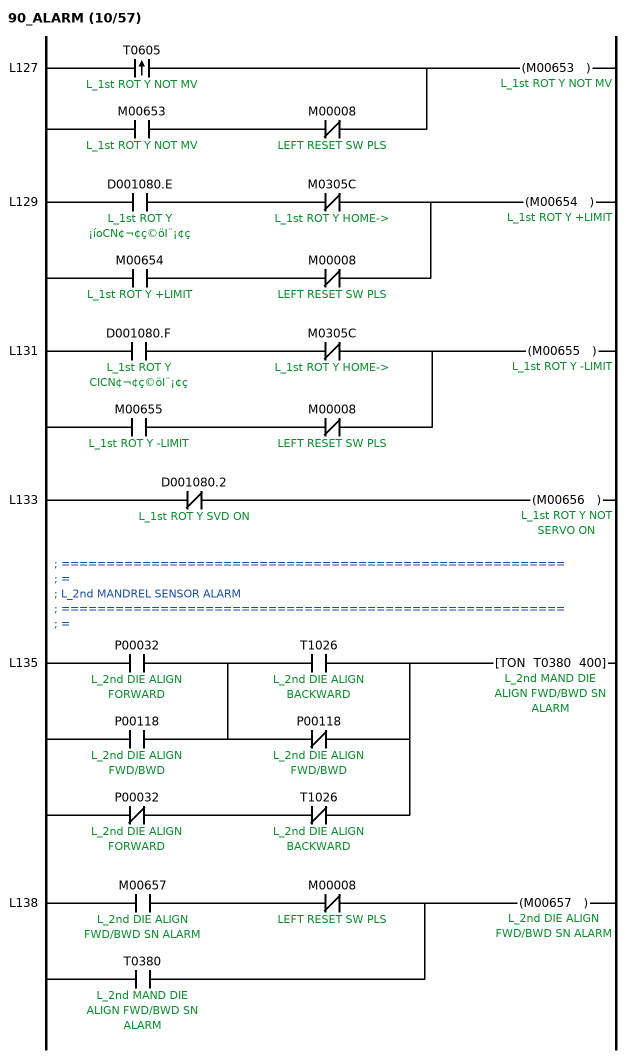
[picture p360: 90_ALARM rungs L127-L138]
; L127
LOADP     T0605	// L_1st ROT Y NOT MV
LOAD      M00653	// L_1st ROT Y NOT MV
AND NOT   M00008	// LEFT RESET SW PLS
OR LOAD
OUT       M00653	// L_1st ROT Y NOT MV
; L129
LOAD      D001080.E	// L_1st ROT Y ¡íoCN¢¬¢ç©öI¨¡¢ç
AND NOT   M0305C	// L_1st ROT Y HOME->
LOAD      M00654	// L_1st ROT Y +LIMIT
AND NOT   M00008	// LEFT RESET SW PLS
OR LOAD
OUT       M00654	// L_1st ROT Y +LIMIT
; L131
LOAD      D001080.F	// L_1st ROT Y CICN¢¬¢ç©öI¨¡¢ç
AND NOT   M0305C	// L_1st ROT Y HOME->
LOAD      M00655	// L_1st ROT Y -LIMIT
AND NOT   M00008	// LEFT RESET SW PLS
OR LOAD
OUT       M00655	// L_1st ROT Y -LIMIT
; L133
LOAD NOT  D001080.2	// L_1st ROT Y SVD ON
OUT       M00656	// L_1st ROT Y NOT SERVO ON
// =========================================================
// 
//        L_2nd MANDREL SENSOR ALARM
// 
// =========================================================
; L135
LOAD      P00032	// L_2nd DIE ALIGN FORWARD
OR        P00118	// L_2nd DIE ALIGN FWD/BWD
LOAD      T1026	// L_2nd DIE ALIGN BACKWARD
OR NOT    P00118	// L_2nd DIE ALIGN FWD/BWD
AND LOAD
LOAD NOT  P00032	// L_2nd DIE ALIGN FORWARD
AND NOT   T1026	// L_2nd DIE ALIGN BACKWARD
OR LOAD
TON       T0380 400	// L_2nd MAND DIE ALIGN FWD/BWD SN ALARM
; L138
LOAD      M00657	// L_2nd DIE ALIGN FWD/BWD SN ALARM
AND NOT   M00008	// LEFT RESET SW PLS
OR        T0380	// L_2nd MAND DIE ALIGN FWD/BWD SN ALARM
OUT       M00657	// L_2nd DIE ALIGN FWD/BWD SN ALARM

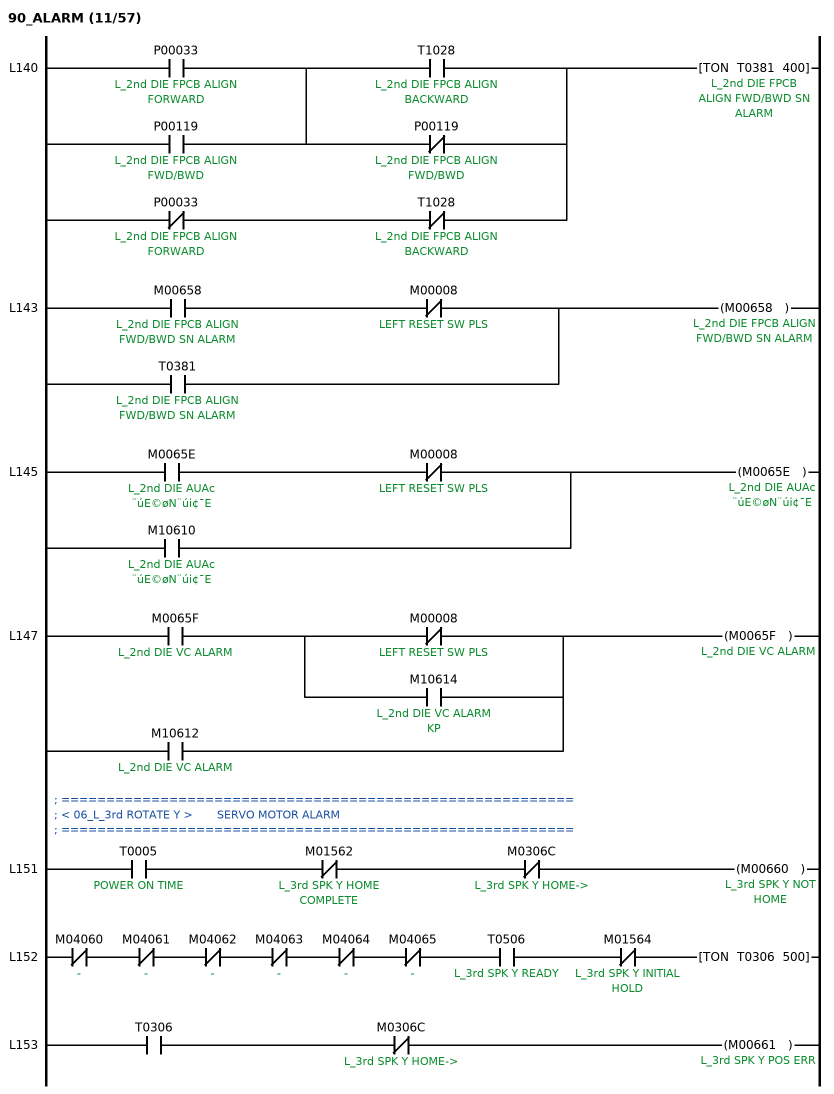
; L140
LOAD      P00033	// L_2nd DIE FPCB ALIGN FORWARD
OR        P00119	// L_2nd DIE FPCB ALIGN FWD/BWD
LOAD      T1028	// L_2nd DIE FPCB ALIGN BACKWARD
OR NOT    P00119	// L_2nd DIE FPCB ALIGN FWD/BWD
AND LOAD
LOAD NOT  P00033	// L_2nd DIE FPCB ALIGN FORWARD
AND NOT   T1028	// L_2nd DIE FPCB ALIGN BACKWARD
OR LOAD
TON       T0381 400	// L_2nd DIE FPCB ALIGN FWD/BWD SN ALARM
; L143
LOAD      M00658	// L_2nd DIE FPCB ALIGN FWD/BWD SN ALARM
AND NOT   M00008	// LEFT RESET SW PLS
OR        T0381	// L_2nd DIE FPCB ALIGN FWD/BWD SN ALARM
OUT       M00658	// L_2nd DIE FPCB ALIGN FWD/BWD SN ALARM
; L145
LOAD      M0065E	// L_2nd DIE AUAc ¨úE©øN¨úi¢¯E
AND NOT   M00008	// LEFT RESET SW PLS
OR        M10610	// L_2nd DIE AUAc ¨úE©øN¨úi¢¯E
OUT       M0065E	// L_2nd DIE AUAc ¨úE©øN¨úi¢¯E
; L147
LOAD      M0065F	// L_2nd DIE VC ALARM
LOAD NOT  M00008	// LEFT RESET SW PLS
OR        M10614	// L_2nd DIE VC ALARM KP
AND LOAD
OR        M10612	// L_2nd DIE VC ALARM
OUT       M0065F	// L_2nd DIE VC ALARM
// =========================================================
// 
//        < 06_L_3rd ROTATE Y >       SERVO MOTOR ALARM
// 
// =========================================================
; L151
LOAD      T0005	// POWER ON TIME
AND NOT   M01562	// L_3rd SPK Y HOME COMPLETE
AND NOT   M0306C	// L_3rd SPK Y HOME->
OUT       M00660	// L_3rd SPK Y NOT HOME
; L152
LOAD NOT  M04060	// -
AND NOT   M04061	// -
AND NOT   M04062	// -
AND NOT   M04063	// -
AND NOT   M04064	// -
AND NOT   M04065	// -
AND       T0506	// L_3rd SPK Y READY
AND NOT   M01564	// L_3rd SPK Y INITIAL HOLD
TON       T0306 500
; L153
LOAD      T0306
AND NOT   M0306C	// L_3rd SPK Y HOME->
OUT       M00661	// L_3rd SPK Y POS ERR

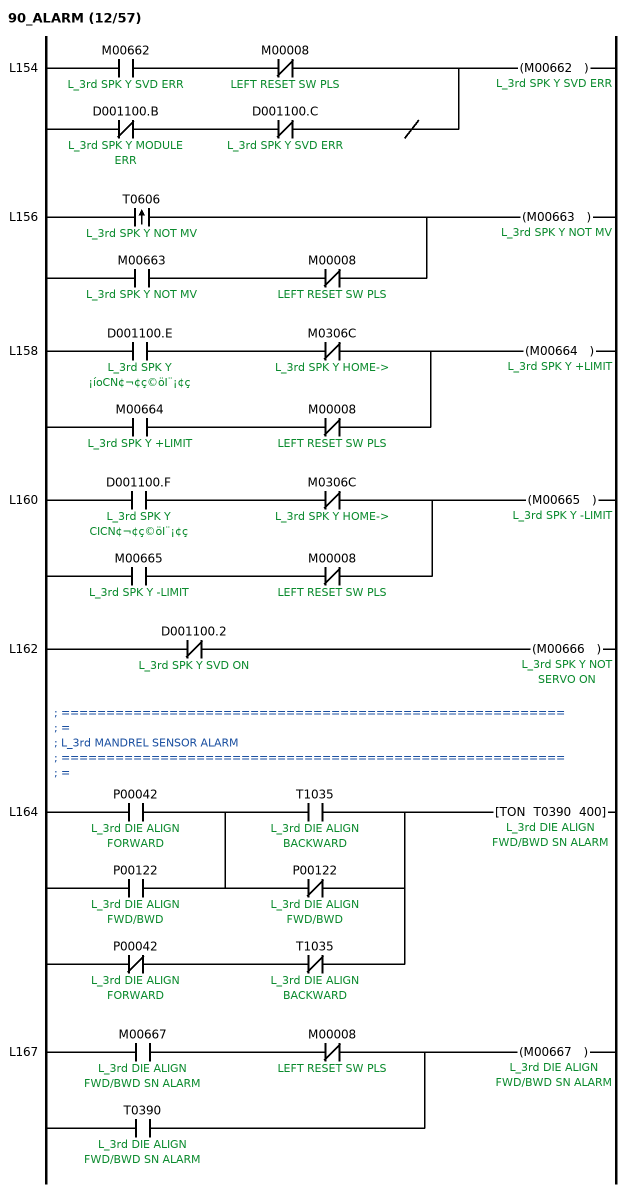
; L154
LOAD      M00662	// L_3rd SPK Y SVD ERR
AND NOT   M00008	// LEFT RESET SW PLS
LOAD NOT  D001100.B	// L_3rd SPK Y MODULE ERR
AND NOT   D001100.C	// L_3rd SPK Y SVD ERR
NOT
OR LOAD
OUT       M00662	// L_3rd SPK Y SVD ERR
; L156
LOADP     T0606	// L_3rd SPK Y NOT MV
LOAD      M00663	// L_3rd SPK Y NOT MV
AND NOT   M00008	// LEFT RESET SW PLS
OR LOAD
OUT       M00663	// L_3rd SPK Y NOT MV
; L158
LOAD      D001100.E	// L_3rd SPK Y ¡íoCN¢¬¢ç©öI¨¡¢ç
AND NOT   M0306C	// L_3rd SPK Y HOME->
LOAD      M00664	// L_3rd SPK Y +LIMIT
AND NOT   M00008	// LEFT RESET SW PLS
OR LOAD
OUT       M00664	// L_3rd SPK Y +LIMIT
; L160
LOAD      D001100.F	// L_3rd SPK Y CICN¢¬¢ç©öI¨¡¢ç
AND NOT   M0306C	// L_3rd SPK Y HOME->
LOAD      M00665	// L_3rd SPK Y -LIMIT
AND NOT   M00008	// LEFT RESET SW PLS
OR LOAD
OUT       M00665	// L_3rd SPK Y -LIMIT
; L162
LOAD NOT  D001100.2	// L_3rd SPK Y SVD ON
OUT       M00666	// L_3rd SPK Y NOT SERVO ON
// =========================================================
// 
//        L_3rd MANDREL SENSOR ALARM
// 
// =========================================================
; L164
LOAD      P00042	// L_3rd DIE ALIGN FORWARD
OR        P00122	// L_3rd DIE ALIGN FWD/BWD
LOAD      T1035	// L_3rd DIE ALIGN BACKWARD
OR NOT    P00122	// L_3rd DIE ALIGN FWD/BWD
AND LOAD
LOAD NOT  P00042	// L_3rd DIE ALIGN FORWARD
AND NOT   T1035	// L_3rd DIE ALIGN BACKWARD
OR LOAD
TON       T0390 400	// L_3rd DIE ALIGN FWD/BWD SN ALARM
; L167
LOAD      M00667	// L_3rd DIE ALIGN FWD/BWD SN ALARM
AND NOT   M00008	// LEFT RESET SW PLS
OR        T0390	// L_3rd DIE ALIGN FWD/BWD SN ALARM
OUT       M00667	// L_3rd DIE ALIGN FWD/BWD SN ALARM

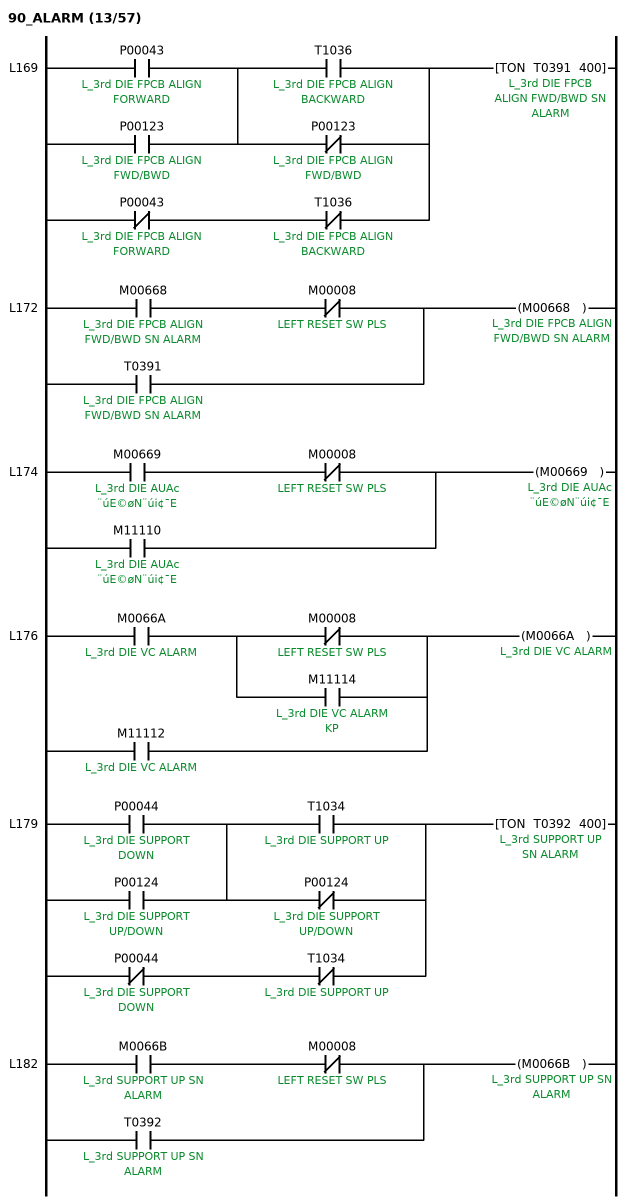
; L169
LOAD      P00043	// L_3rd DIE FPCB ALIGN FORWARD
OR        P00123	// L_3rd DIE FPCB ALIGN FWD/BWD
LOAD      T1036	// L_3rd DIE FPCB ALIGN BACKWARD
OR NOT    P00123	// L_3rd DIE FPCB ALIGN FWD/BWD
AND LOAD
LOAD NOT  P00043	// L_3rd DIE FPCB ALIGN FORWARD
AND NOT   T1036	// L_3rd DIE FPCB ALIGN BACKWARD
OR LOAD
TON       T0391 400	// L_3rd DIE FPCB ALIGN FWD/BWD SN ALARM
; L172
LOAD      M00668	// L_3rd DIE FPCB ALIGN FWD/BWD SN ALARM
AND NOT   M00008	// LEFT RESET SW PLS
OR        T0391	// L_3rd DIE FPCB ALIGN FWD/BWD SN ALARM
OUT       M00668	// L_3rd DIE FPCB ALIGN FWD/BWD SN ALARM
; L174
LOAD      M00669	// L_3rd DIE AUAc ¨úE©øN¨úi¢¯E
AND NOT   M00008	// LEFT RESET SW PLS
OR        M11110	// L_3rd DIE AUAc ¨úE©øN¨úi¢¯E
OUT       M00669	// L_3rd DIE AUAc ¨úE©øN¨úi¢¯E
; L176
LOAD      M0066A	// L_3rd DIE VC ALARM
LOAD NOT  M00008	// LEFT RESET SW PLS
OR        M11114	// L_3rd DIE VC ALARM KP
AND LOAD
OR        M11112	// L_3rd DIE VC ALARM
OUT       M0066A	// L_3rd DIE VC ALARM
; L179
LOAD      P00044	// L_3rd DIE SUPPORT DOWN
OR        P00124	// L_3rd DIE SUPPORT UP/DOWN
LOAD      T1034	// L_3rd DIE SUPPORT UP
OR NOT    P00124	// L_3rd DIE SUPPORT UP/DOWN
AND LOAD
LOAD NOT  P00044	// L_3rd DIE SUPPORT DOWN
AND NOT   T1034	// L_3rd DIE SUPPORT UP
OR LOAD
TON       T0392 400	// L_3rd SUPPORT UP SN ALARM
; L182
LOAD      M0066B	// L_3rd SUPPORT UP SN ALARM
AND NOT   M00008	// LEFT RESET SW PLS
OR        T0392	// L_3rd SUPPORT UP SN ALARM
OUT       M0066B	// L_3rd SUPPORT UP SN ALARM

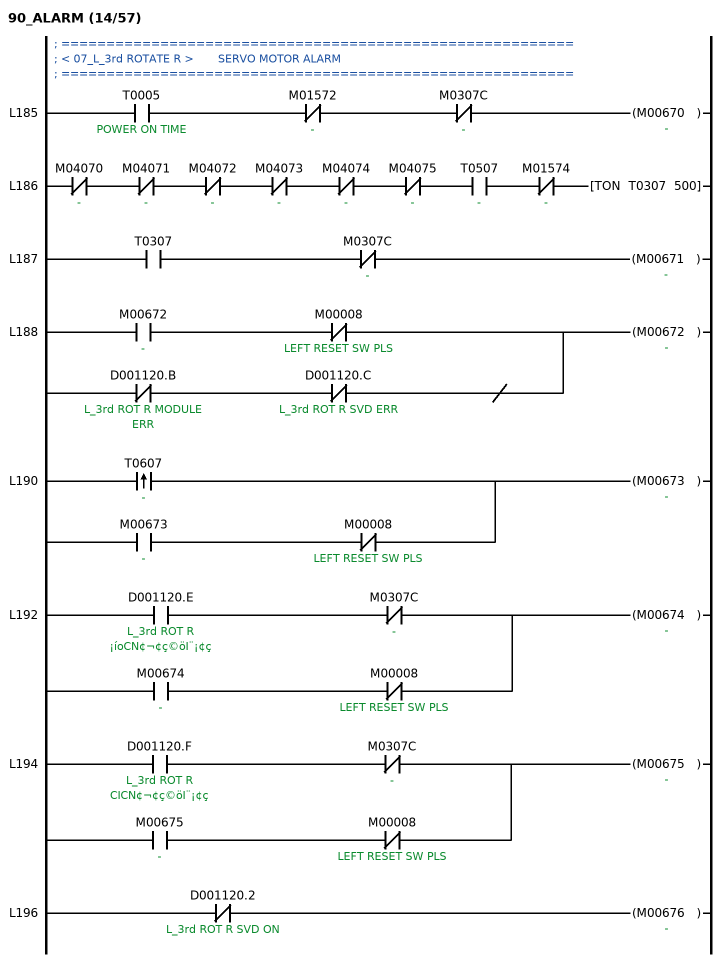
// =========================================================
// 
//        < 07_L_3rd ROTATE R >       SERVO MOTOR ALARM
// 
// =========================================================
; L185
LOAD      T0005	// POWER ON TIME
AND NOT   M01572	// -
AND NOT   M0307C	// -
OUT       M00670	// -
; L186
LOAD NOT  M04070	// -
AND NOT   M04071	// -
AND NOT   M04072	// -
AND NOT   M04073	// -
AND NOT   M04074	// -
AND NOT   M04075	// -
AND       T0507	// -
AND NOT   M01574	// -
TON       T0307 500
; L187
LOAD      T0307
AND NOT   M0307C	// -
OUT       M00671	// -
; L188
LOAD      M00672	// -
AND NOT   M00008	// LEFT RESET SW PLS
LOAD NOT  D001120.B	// L_3rd ROT R MODULE ERR
AND NOT   D001120.C	// L_3rd ROT R SVD ERR
NOT
OR LOAD
OUT       M00672	// -
; L190
LOADP     T0607	// -
LOAD      M00673	// -
AND NOT   M00008	// LEFT RESET SW PLS
OR LOAD
OUT       M00673	// -
; L192
LOAD      D001120.E	// L_3rd ROT R ¡íoCN¢¬¢ç©öI¨¡¢ç
AND NOT   M0307C	// -
LOAD      M00674	// -
AND NOT   M00008	// LEFT RESET SW PLS
OR LOAD
OUT       M00674	// -
; L194
LOAD      D001120.F	// L_3rd ROT R CICN¢¬¢ç©öI¨¡¢ç
AND NOT   M0307C	// -
LOAD      M00675	// -
AND NOT   M00008	// LEFT RESET SW PLS
OR LOAD
OUT       M00675	// -
; L196
LOAD NOT  D001120.2	// L_3rd ROT R SVD ON
OUT       M00676	// -

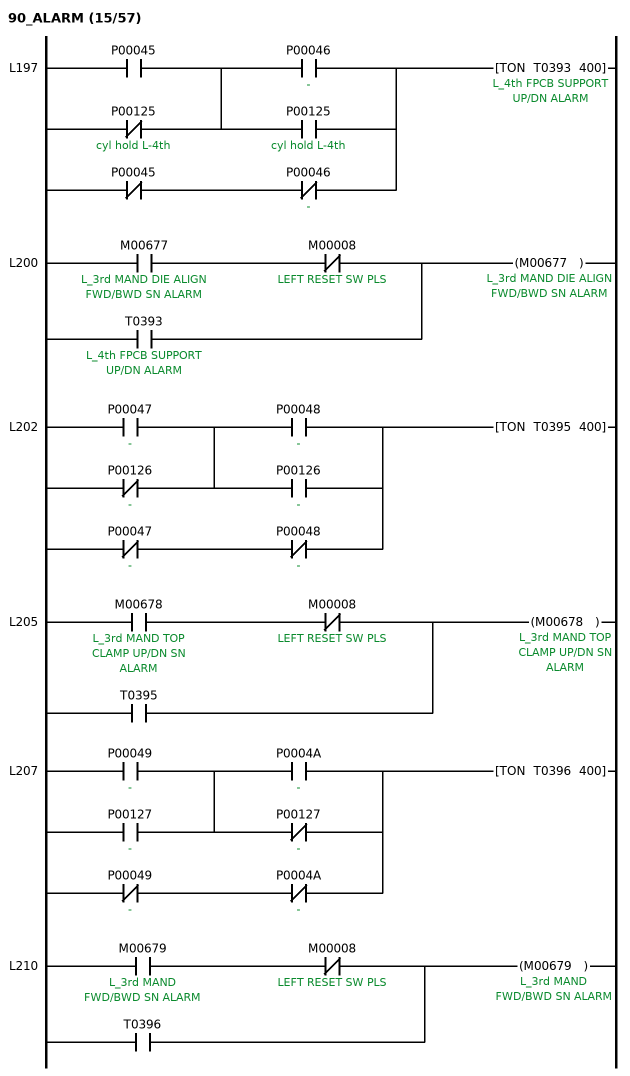
; L197
LOAD      P00045
OR NOT    P00125	// cyl hold L-4th
LOAD      P00046	// -
OR        P00125	// cyl hold L-4th
AND LOAD
LOAD NOT  P00045
AND NOT   P00046	// -
OR LOAD
TON       T0393 400	// L_4th FPCB SUPPORT UP/DN ALARM
; L200
LOAD      M00677	// L_3rd MAND DIE ALIGN FWD/BWD SN ALARM
AND NOT   M00008	// LEFT RESET SW PLS
OR        T0393	// L_4th FPCB SUPPORT UP/DN ALARM
OUT       M00677	// L_3rd MAND DIE ALIGN FWD/BWD SN ALARM
; L202
LOAD      P00047	// -
OR NOT    P00126	// -
LOAD      P00048	// -
OR        P00126	// -
AND LOAD
LOAD NOT  P00047	// -
AND NOT   P00048	// -
OR LOAD
TON       T0395 400
; L205
LOAD      M00678	// L_3rd MAND TOP CLAMP UP/DN SN ALARM
AND NOT   M00008	// LEFT RESET SW PLS
OR        T0395
OUT       M00678	// L_3rd MAND TOP CLAMP UP/DN SN ALARM
; L207
LOAD      P00049	// -
OR        P00127	// -
LOAD      P0004A	// -
OR NOT    P00127	// -
AND LOAD
LOAD NOT  P00049	// -
AND NOT   P0004A	// -
OR LOAD
TON       T0396 400
; L210
LOAD      M00679	// L_3rd MAND FWD/BWD SN ALARM
AND NOT   M00008	// LEFT RESET SW PLS
OR        T0396
OUT       M00679	// L_3rd MAND FWD/BWD SN ALARM

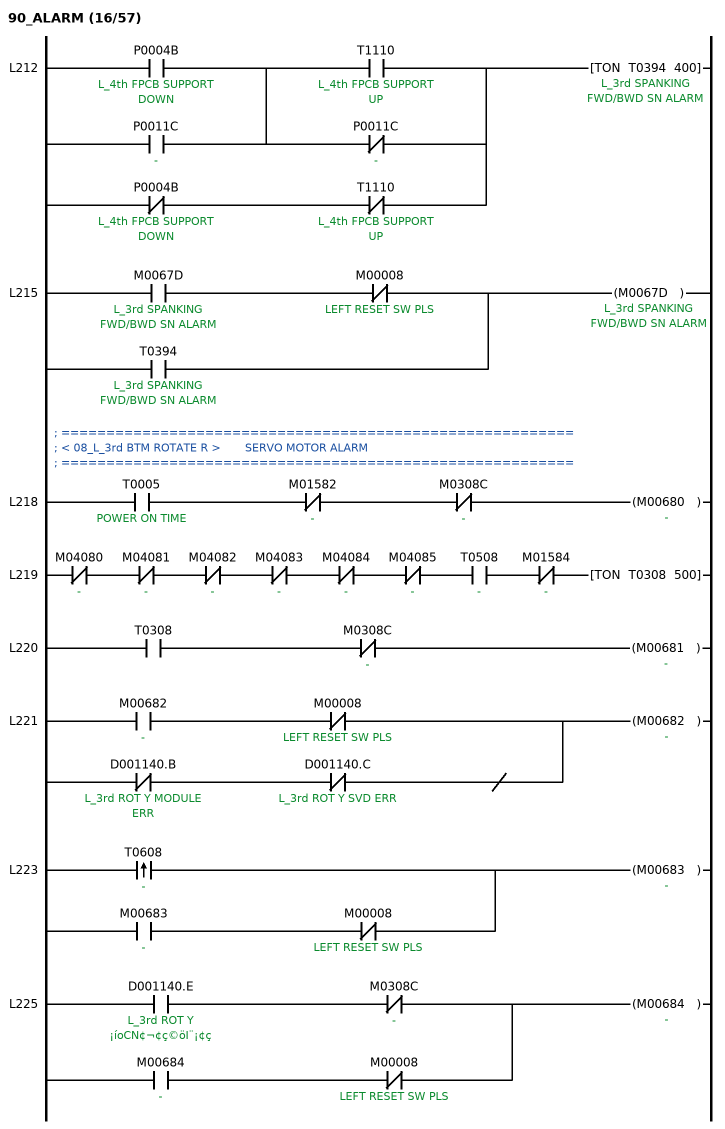
; L212
LOAD      P0004B	// L_4th FPCB SUPPORT DOWN
OR        P0011C	// -
LOAD      T1110	// L_4th FPCB SUPPORT UP
OR NOT    P0011C	// -
AND LOAD
LOAD NOT  P0004B	// L_4th FPCB SUPPORT DOWN
AND NOT   T1110	// L_4th FPCB SUPPORT UP
OR LOAD
TON       T0394 400	// L_3rd SPANKING FWD/BWD SN ALARM
; L215
LOAD      M0067D	// L_3rd SPANKING FWD/BWD SN ALARM
AND NOT   M00008	// LEFT RESET SW PLS
OR        T0394	// L_3rd SPANKING FWD/BWD SN ALARM
OUT       M0067D	// L_3rd SPANKING FWD/BWD SN ALARM
// =========================================================
// 
//        < 08_L_3rd BTM ROTATE R >       SERVO MOTOR ALARM
// 
// =========================================================
; L218
LOAD      T0005	// POWER ON TIME
AND NOT   M01582	// -
AND NOT   M0308C	// -
OUT       M00680	// -
; L219
LOAD NOT  M04080	// -
AND NOT   M04081	// -
AND NOT   M04082	// -
AND NOT   M04083	// -
AND NOT   M04084	// -
AND NOT   M04085	// -
AND       T0508	// -
AND NOT   M01584	// -
TON       T0308 500
; L220
LOAD      T0308
AND NOT   M0308C	// -
OUT       M00681	// -
; L221
LOAD      M00682	// -
AND NOT   M00008	// LEFT RESET SW PLS
LOAD NOT  D001140.B	// L_3rd ROT Y MODULE ERR
AND NOT   D001140.C	// L_3rd ROT Y SVD ERR
NOT
OR LOAD
OUT       M00682	// -
; L223
LOADP     T0608	// -
LOAD      M00683	// -
AND NOT   M00008	// LEFT RESET SW PLS
OR LOAD
OUT       M00683	// -
; L225
LOAD      D001140.E	// L_3rd ROT Y ¡íoCN¢¬¢ç©öI¨¡¢ç
AND NOT   M0308C	// -
LOAD      M00684	// -
AND NOT   M00008	// LEFT RESET SW PLS
OR LOAD
OUT       M00684	// -

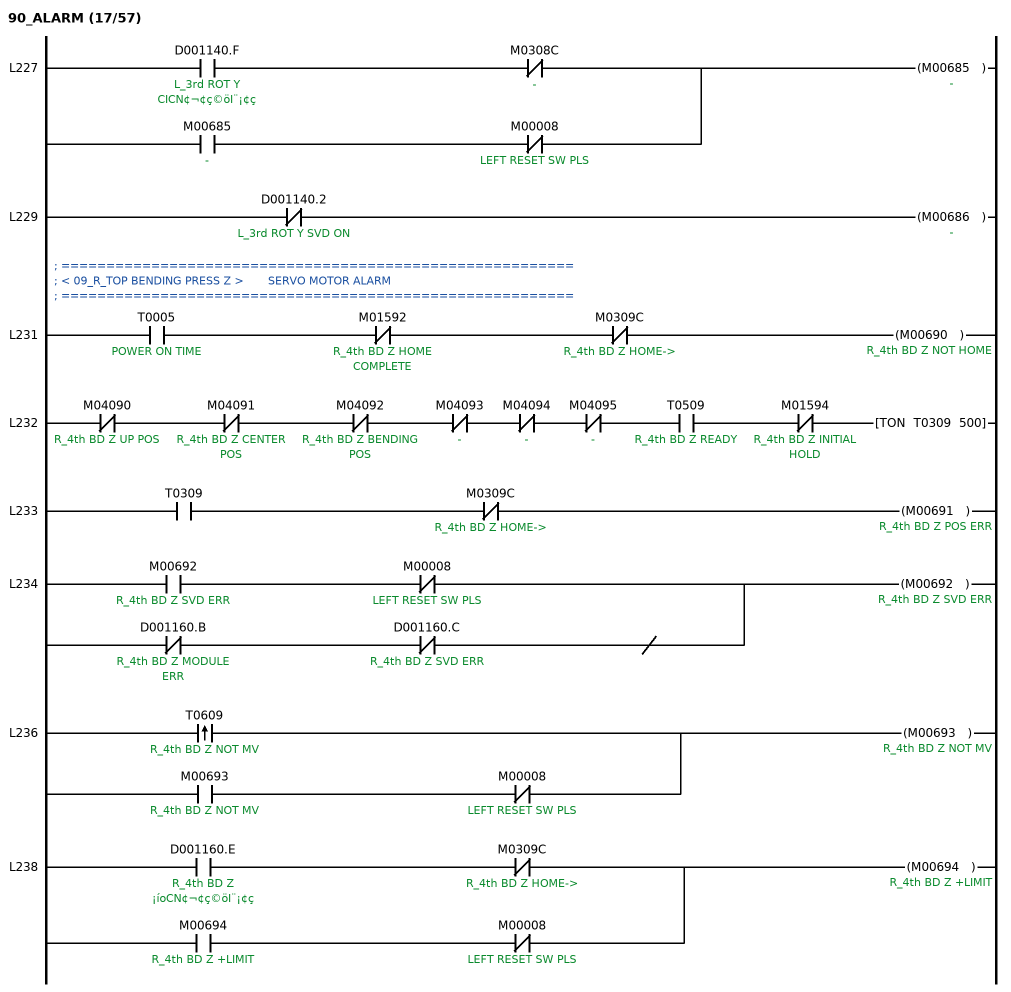
; L227
LOAD      D001140.F	// L_3rd ROT Y CICN¢¬¢ç©öI¨¡¢ç
AND NOT   M0308C	// -
LOAD      M00685	// -
AND NOT   M00008	// LEFT RESET SW PLS
OR LOAD
OUT       M00685	// -
; L229
LOAD NOT  D001140.2	// L_3rd ROT Y SVD ON
OUT       M00686	// -
// =========================================================
// 
//        < 09_R_TOP BENDING PRESS Z >       SERVO MOTOR ALARM
// 
// =========================================================
; L231
LOAD      T0005	// POWER ON TIME
AND NOT   M01592	// R_4th BD Z HOME COMPLETE
AND NOT   M0309C	// R_4th BD Z HOME->
OUT       M00690	// R_4th BD Z NOT HOME
; L232
LOAD NOT  M04090	// R_4th BD Z UP POS
AND NOT   M04091	// R_4th BD Z CENTER POS
AND NOT   M04092	// R_4th BD Z BENDING POS
AND NOT   M04093	// -
AND NOT   M04094	// -
AND NOT   M04095	// -
AND       T0509	// R_4th BD Z READY
AND NOT   M01594	// R_4th BD Z INITIAL HOLD
TON       T0309 500
; L233
LOAD      T0309
AND NOT   M0309C	// R_4th BD Z HOME->
OUT       M00691	// R_4th BD Z POS ERR
; L234
LOAD      M00692	// R_4th BD Z SVD ERR
AND NOT   M00008	// LEFT RESET SW PLS
LOAD NOT  D001160.B	// R_4th BD Z MODULE ERR
AND NOT   D001160.C	// R_4th BD Z SVD ERR
NOT
OR LOAD
OUT       M00692	// R_4th BD Z SVD ERR
; L236
LOADP     T0609	// R_4th BD Z NOT MV
LOAD      M00693	// R_4th BD Z NOT MV
AND NOT   M00008	// LEFT RESET SW PLS
OR LOAD
OUT       M00693	// R_4th BD Z NOT MV
; L238
LOAD      D001160.E	// R_4th BD Z ¡íoCN¢¬¢ç©öI¨¡¢ç
AND NOT   M0309C	// R_4th BD Z HOME->
LOAD      M00694	// R_4th BD Z +LIMIT
AND NOT   M00008	// LEFT RESET SW PLS
OR LOAD
OUT       M00694	// R_4th BD Z +LIMIT

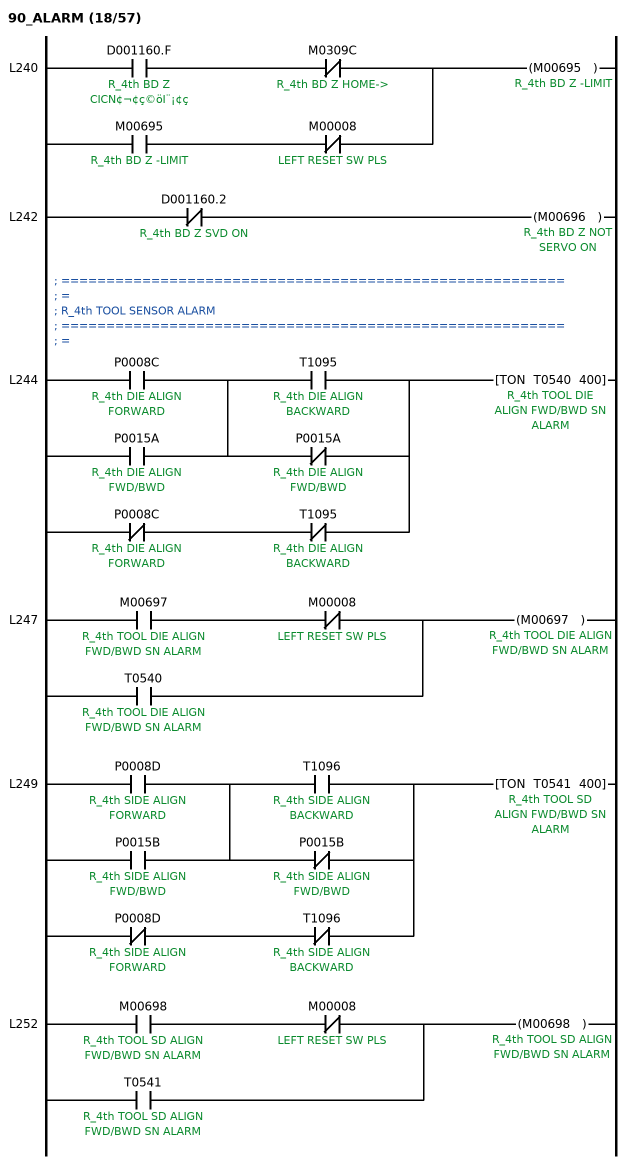
; L240
LOAD      D001160.F	// R_4th BD Z CICN¢¬¢ç©öI¨¡¢ç
AND NOT   M0309C	// R_4th BD Z HOME->
LOAD      M00695	// R_4th BD Z -LIMIT
AND NOT   M00008	// LEFT RESET SW PLS
OR LOAD
OUT       M00695	// R_4th BD Z -LIMIT
; L242
LOAD NOT  D001160.2	// R_4th BD Z SVD ON
OUT       M00696	// R_4th BD Z NOT SERVO ON
// =========================================================
// 
//        R_4th TOOL SENSOR ALARM
// 
// =========================================================
; L244
LOAD      P0008C	// R_4th DIE ALIGN FORWARD
OR        P0015A	// R_4th DIE ALIGN FWD/BWD
LOAD      T1095	// R_4th DIE ALIGN BACKWARD
OR NOT    P0015A	// R_4th DIE ALIGN FWD/BWD
AND LOAD
LOAD NOT  P0008C	// R_4th DIE ALIGN FORWARD
AND NOT   T1095	// R_4th DIE ALIGN BACKWARD
OR LOAD
TON       T0540 400	// R_4th TOOL DIE ALIGN FWD/BWD SN ALARM
; L247
LOAD      M00697	// R_4th TOOL DIE ALIGN FWD/BWD SN ALARM
AND NOT   M00008	// LEFT RESET SW PLS
OR        T0540	// R_4th TOOL DIE ALIGN FWD/BWD SN ALARM
OUT       M00697	// R_4th TOOL DIE ALIGN FWD/BWD SN ALARM
; L249
LOAD      P0008D	// R_4th SIDE ALIGN FORWARD
OR        P0015B	// R_4th SIDE ALIGN FWD/BWD
LOAD      T1096	// R_4th SIDE ALIGN BACKWARD
OR NOT    P0015B	// R_4th SIDE ALIGN FWD/BWD
AND LOAD
LOAD NOT  P0008D	// R_4th SIDE ALIGN FORWARD
AND NOT   T1096	// R_4th SIDE ALIGN BACKWARD
OR LOAD
TON       T0541 400	// R_4th TOOL SD ALIGN FWD/BWD SN ALARM
; L252
LOAD      M00698	// R_4th TOOL SD ALIGN FWD/BWD SN ALARM
AND NOT   M00008	// LEFT RESET SW PLS
OR        T0541	// R_4th TOOL SD ALIGN FWD/BWD SN ALARM
OUT       M00698	// R_4th TOOL SD ALIGN FWD/BWD SN ALARM

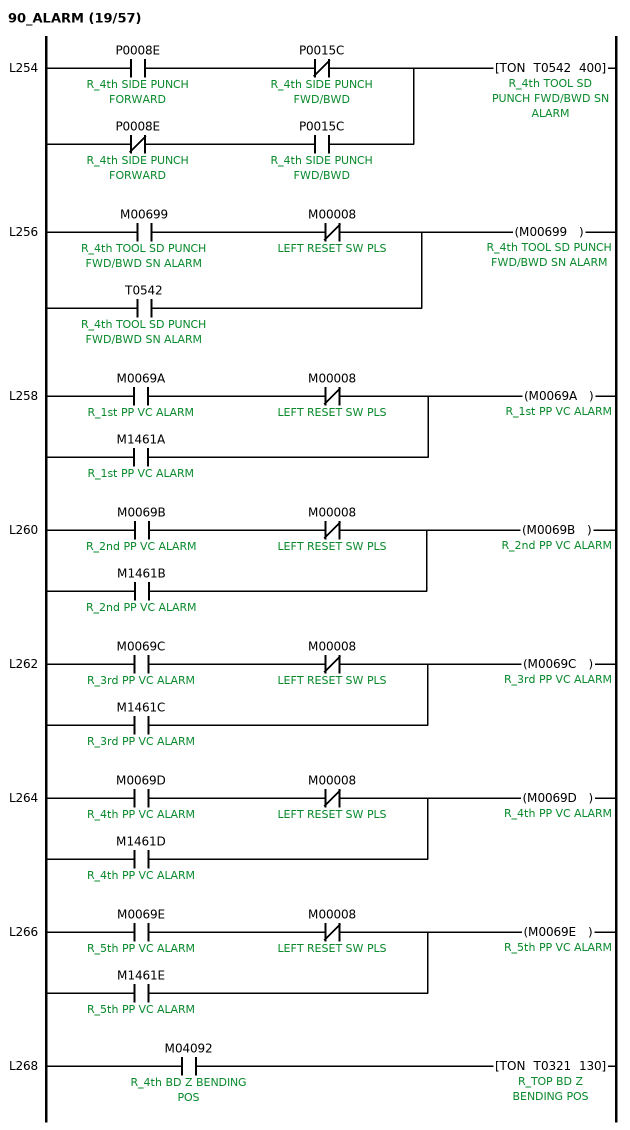
; L254
LOAD      P0008E	// R_4th SIDE PUNCH FORWARD
AND NOT   P0015C	// R_4th SIDE PUNCH FWD/BWD
LOAD NOT  P0008E	// R_4th SIDE PUNCH FORWARD
AND       P0015C	// R_4th SIDE PUNCH FWD/BWD
OR LOAD
TON       T0542 400	// R_4th TOOL SD PUNCH FWD/BWD SN ALARM
; L256
LOAD      M00699	// R_4th TOOL SD PUNCH FWD/BWD SN ALARM
AND NOT   M00008	// LEFT RESET SW PLS
OR        T0542	// R_4th TOOL SD PUNCH FWD/BWD SN ALARM
OUT       M00699	// R_4th TOOL SD PUNCH FWD/BWD SN ALARM
; L258
LOAD      M0069A	// R_1st PP VC ALARM
AND NOT   M00008	// LEFT RESET SW PLS
OR        M1461A	// R_1st PP VC ALARM
OUT       M0069A	// R_1st PP VC ALARM
; L260
LOAD      M0069B	// R_2nd PP VC ALARM
AND NOT   M00008	// LEFT RESET SW PLS
OR        M1461B	// R_2nd PP VC ALARM
OUT       M0069B	// R_2nd PP VC ALARM
; L262
LOAD      M0069C	// R_3rd PP VC ALARM
AND NOT   M00008	// LEFT RESET SW PLS
OR        M1461C	// R_3rd PP VC ALARM
OUT       M0069C	// R_3rd PP VC ALARM
; L264
LOAD      M0069D	// R_4th PP VC ALARM
AND NOT   M00008	// LEFT RESET SW PLS
OR        M1461D	// R_4th PP VC ALARM
OUT       M0069D	// R_4th PP VC ALARM
; L266
LOAD      M0069E	// R_5th PP VC ALARM
AND NOT   M00008	// LEFT RESET SW PLS
OR        M1461E	// R_5th PP VC ALARM
OUT       M0069E	// R_5th PP VC ALARM
; L268
LOAD      M04092	// R_4th BD Z BENDING POS
TON       T0321 130	// R_TOP BD Z BENDING POS

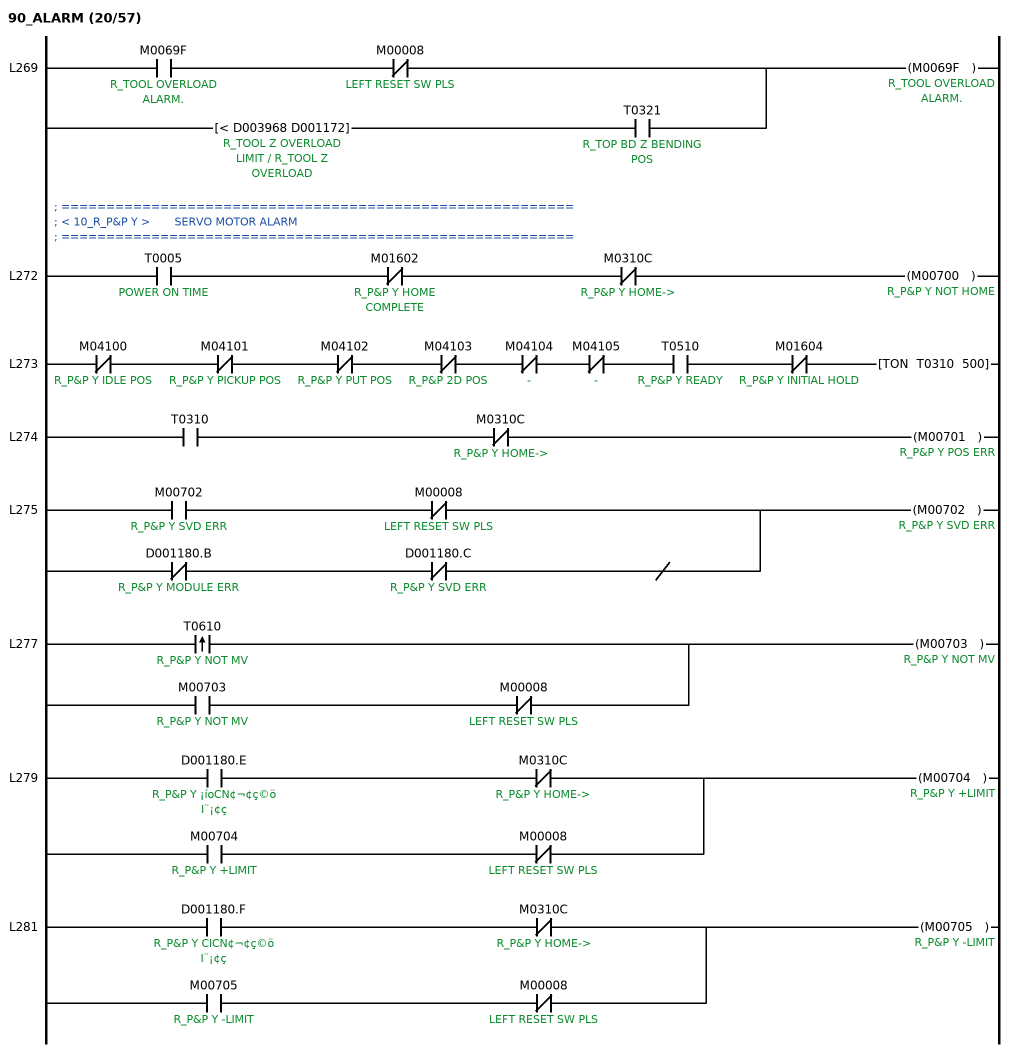
; L269
LOAD      M0069F	// R_TOOL OVERLOAD ALARM.
AND NOT   M00008	// LEFT RESET SW PLS
LOAD<     D003968 D001172	// R_TOOL Z OVERLOAD LIMIT / R_TOOL Z OVERLOAD
AND       T0321	// R_TOP BD Z BENDING POS
OR LOAD
OUT       M0069F	// R_TOOL OVERLOAD ALARM.
// =========================================================
// 
//        < 10_R_P&P Y >       SERVO MOTOR ALARM
// 
// =========================================================
; L272
LOAD      T0005	// POWER ON TIME
AND NOT   M01602	// R_P&P Y HOME COMPLETE
AND NOT   M0310C	// R_P&P Y HOME->
OUT       M00700	// R_P&P Y NOT HOME
; L273
LOAD NOT  M04100	// R_P&P Y IDLE POS
AND NOT   M04101	// R_P&P Y PICKUP POS
AND NOT   M04102	// R_P&P Y PUT POS
AND NOT   M04103	// R_P&P 2D POS
AND NOT   M04104	// -
AND NOT   M04105	// -
AND       T0510	// R_P&P Y READY
AND NOT   M01604	// R_P&P Y INITIAL HOLD
TON       T0310 500
; L274
LOAD      T0310
AND NOT   M0310C	// R_P&P Y HOME->
OUT       M00701	// R_P&P Y POS ERR
; L275
LOAD      M00702	// R_P&P Y SVD ERR
AND NOT   M00008	// LEFT RESET SW PLS
LOAD NOT  D001180.B	// R_P&P Y MODULE ERR
AND NOT   D001180.C	// R_P&P Y SVD ERR
NOT
OR LOAD
OUT       M00702	// R_P&P Y SVD ERR
; L277
LOADP     T0610	// R_P&P Y NOT MV
LOAD      M00703	// R_P&P Y NOT MV
AND NOT   M00008	// LEFT RESET SW PLS
OR LOAD
OUT       M00703	// R_P&P Y NOT MV
; L279
LOAD      D001180.E	// R_P&P Y ¡íoCN¢¬¢ç©öI¨¡¢ç
AND NOT   M0310C	// R_P&P Y HOME->
LOAD      M00704	// R_P&P Y +LIMIT
AND NOT   M00008	// LEFT RESET SW PLS
OR LOAD
OUT       M00704	// R_P&P Y +LIMIT
; L281
LOAD      D001180.F	// R_P&P Y CICN¢¬¢ç©öI¨¡¢ç
AND NOT   M0310C	// R_P&P Y HOME->
LOAD      M00705	// R_P&P Y -LIMIT
AND NOT   M00008	// LEFT RESET SW PLS
OR LOAD
OUT       M00705	// R_P&P Y -LIMIT

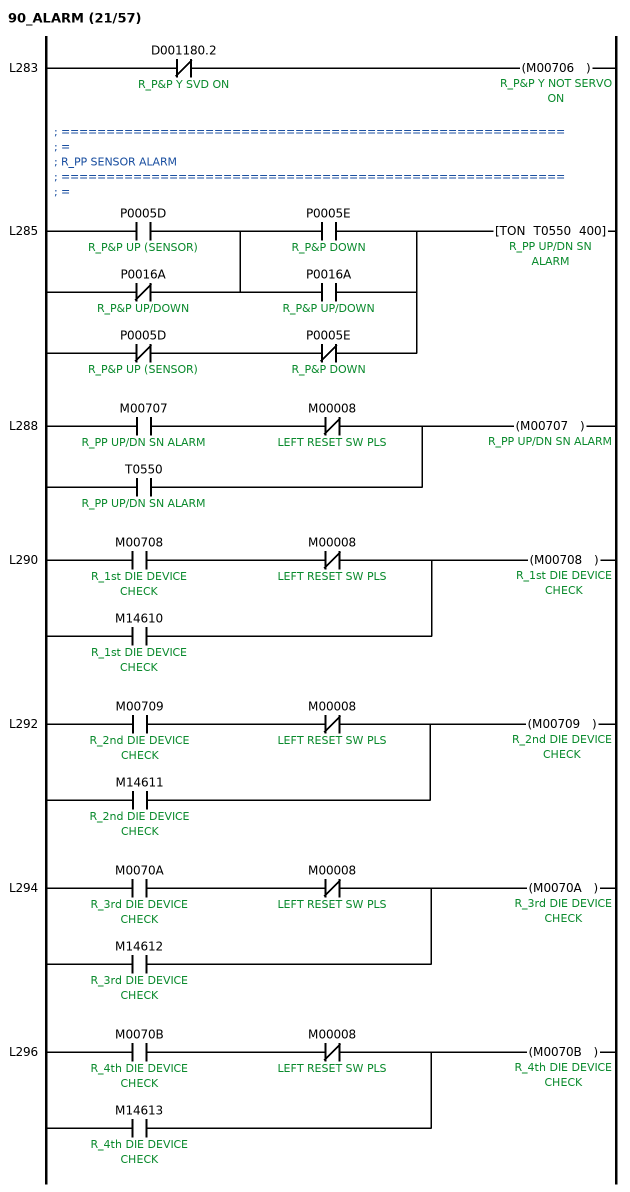
; L283
LOAD NOT  D001180.2	// R_P&P Y SVD ON
OUT       M00706	// R_P&P Y NOT SERVO ON
// =========================================================
// 
//       R_PP SENSOR ALARM
// 
// =========================================================
; L285
LOAD      P0005D	// R_P&P UP (SENSOR)
OR NOT    P0016A	// R_P&P UP/DOWN
LOAD      P0005E	// R_P&P DOWN
OR        P0016A	// R_P&P UP/DOWN
AND LOAD
LOAD NOT  P0005D	// R_P&P UP (SENSOR)
AND NOT   P0005E	// R_P&P DOWN
OR LOAD
TON       T0550 400	// R_PP UP/DN SN ALARM
; L288
LOAD      M00707	// R_PP UP/DN SN ALARM
AND NOT   M00008	// LEFT RESET SW PLS
OR        T0550	// R_PP UP/DN SN ALARM
OUT       M00707	// R_PP UP/DN SN ALARM
; L290
LOAD      M00708	// R_1st DIE DEVICE CHECK
AND NOT   M00008	// LEFT RESET SW PLS
OR        M14610	// R_1st DIE DEVICE CHECK
OUT       M00708	// R_1st DIE DEVICE CHECK
; L292
LOAD      M00709	// R_2nd DIE DEVICE CHECK
AND NOT   M00008	// LEFT RESET SW PLS
OR        M14611	// R_2nd DIE DEVICE CHECK
OUT       M00709	// R_2nd DIE DEVICE CHECK
; L294
LOAD      M0070A	// R_3rd DIE DEVICE CHECK
AND NOT   M00008	// LEFT RESET SW PLS
OR        M14612	// R_3rd DIE DEVICE CHECK
OUT       M0070A	// R_3rd DIE DEVICE CHECK
; L296
LOAD      M0070B	// R_4th DIE DEVICE CHECK
AND NOT   M00008	// LEFT RESET SW PLS
OR        M14613	// R_4th DIE DEVICE CHECK
OUT       M0070B	// R_4th DIE DEVICE CHECK

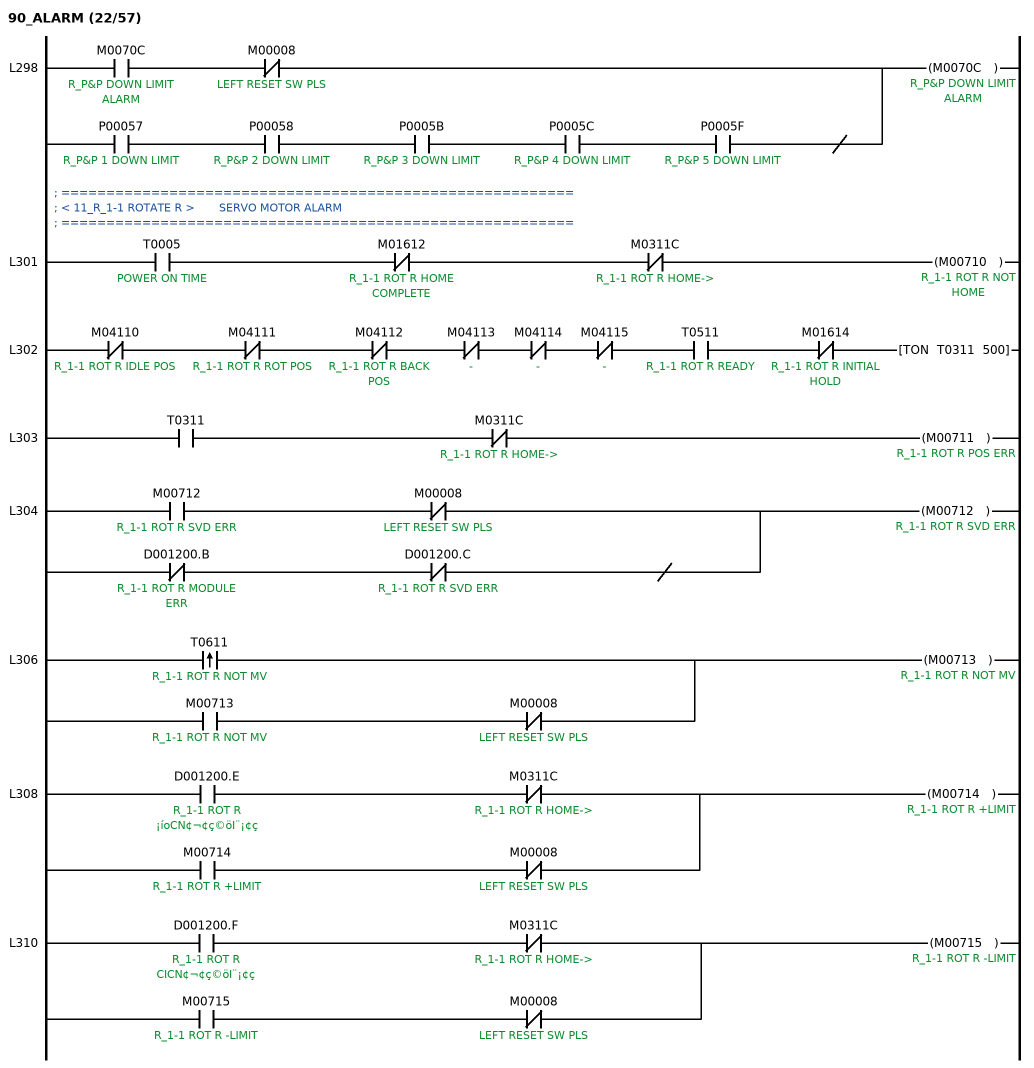
; L298
LOAD      M0070C	// R_P&P DOWN LIMIT ALARM
AND NOT   M00008	// LEFT RESET SW PLS
LOAD      P00057	// R_P&P 1 DOWN LIMIT
AND       P00058	// R_P&P 2 DOWN LIMIT
AND       P0005B	// R_P&P 3 DOWN LIMIT
AND       P0005C	// R_P&P 4 DOWN LIMIT
AND       P0005F	// R_P&P 5 DOWN LIMIT
NOT
OR LOAD
OUT       M0070C	// R_P&P DOWN LIMIT ALARM
// =========================================================
// 
//        < 11_R_1-1 ROTATE R >       SERVO MOTOR ALARM
// 
// =========================================================
; L301
LOAD      T0005	// POWER ON TIME
AND NOT   M01612	// R_1-1 ROT R HOME COMPLETE
AND NOT   M0311C	// R_1-1 ROT R HOME->
OUT       M00710	// R_1-1 ROT R NOT HOME
; L302
LOAD NOT  M04110	// R_1-1 ROT R IDLE POS
AND NOT   M04111	// R_1-1 ROT R ROT POS
AND NOT   M04112	// R_1-1 ROT R BACK POS
AND NOT   M04113	// -
AND NOT   M04114	// -
AND NOT   M04115	// -
AND       T0511	// R_1-1 ROT R READY
AND NOT   M01614	// R_1-1 ROT R INITIAL HOLD
TON       T0311 500
; L303
LOAD      T0311
AND NOT   M0311C	// R_1-1 ROT R HOME->
OUT       M00711	// R_1-1 ROT R POS ERR
; L304
LOAD      M00712	// R_1-1 ROT R SVD ERR
AND NOT   M00008	// LEFT RESET SW PLS
LOAD NOT  D001200.B	// R_1-1 ROT R MODULE ERR
AND NOT   D001200.C	// R_1-1 ROT R SVD ERR
NOT
OR LOAD
OUT       M00712	// R_1-1 ROT R SVD ERR
; L306
LOADP     T0611	// R_1-1 ROT R NOT MV
LOAD      M00713	// R_1-1 ROT R NOT MV
AND NOT   M00008	// LEFT RESET SW PLS
OR LOAD
OUT       M00713	// R_1-1 ROT R NOT MV
; L308
LOAD      D001200.E	// R_1-1 ROT R ¡íoCN¢¬¢ç©öI¨¡¢ç
AND NOT   M0311C	// R_1-1 ROT R HOME->
LOAD      M00714	// R_1-1 ROT R +LIMIT
AND NOT   M00008	// LEFT RESET SW PLS
OR LOAD
OUT       M00714	// R_1-1 ROT R +LIMIT
; L310
LOAD      D001200.F	// R_1-1 ROT R CICN¢¬¢ç©öI¨¡¢ç
AND NOT   M0311C	// R_1-1 ROT R HOME->
LOAD      M00715	// R_1-1 ROT R -LIMIT
AND NOT   M00008	// LEFT RESET SW PLS
OR LOAD
OUT       M00715	// R_1-1 ROT R -LIMIT

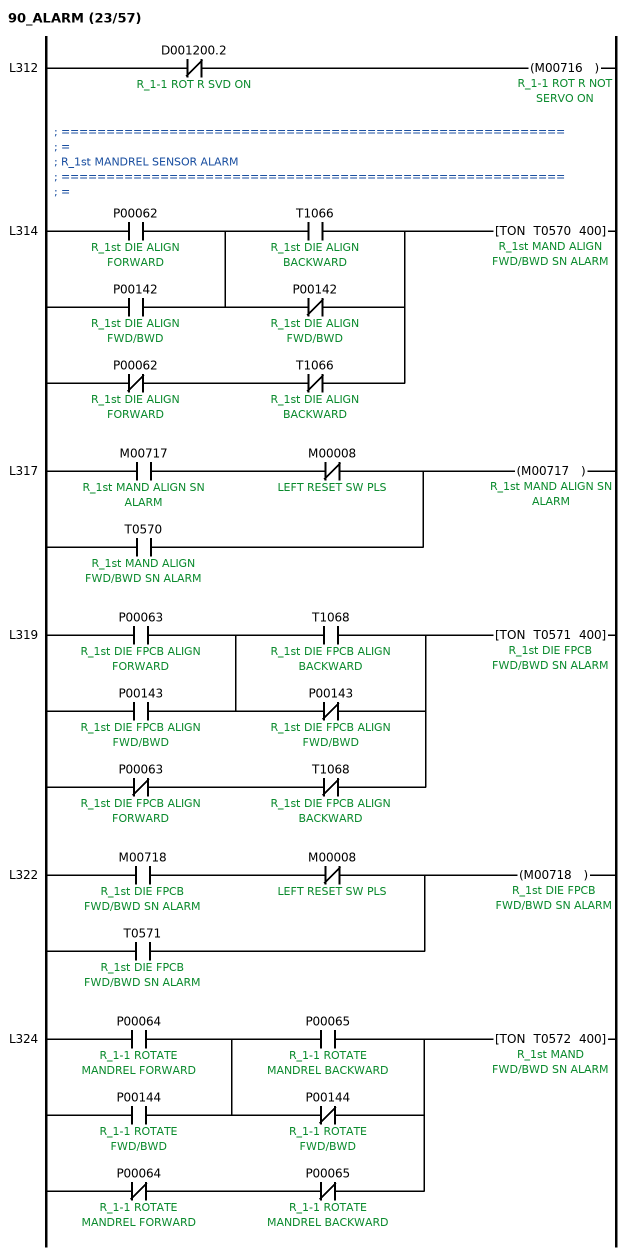
; L312
LOAD NOT  D001200.2	// R_1-1 ROT R SVD ON
OUT       M00716	// R_1-1 ROT R NOT SERVO ON
// =========================================================
// 
//        R_1st MANDREL SENSOR ALARM
// 
// =========================================================
; L314
LOAD      P00062	// R_1st DIE ALIGN FORWARD
OR        P00142	// R_1st DIE ALIGN FWD/BWD
LOAD      T1066	// R_1st DIE ALIGN BACKWARD
OR NOT    P00142	// R_1st DIE ALIGN FWD/BWD
AND LOAD
LOAD NOT  P00062	// R_1st DIE ALIGN FORWARD
AND NOT   T1066	// R_1st DIE ALIGN BACKWARD
OR LOAD
TON       T0570 400	// R_1st MAND ALIGN FWD/BWD SN ALARM
; L317
LOAD      M00717	// R_1st MAND ALIGN SN ALARM
AND NOT   M00008	// LEFT RESET SW PLS
OR        T0570	// R_1st MAND ALIGN FWD/BWD SN ALARM
OUT       M00717	// R_1st MAND ALIGN SN ALARM
; L319
LOAD      P00063	// R_1st DIE FPCB ALIGN FORWARD
OR        P00143	// R_1st DIE FPCB ALIGN FWD/BWD
LOAD      T1068	// R_1st DIE FPCB ALIGN BACKWARD
OR NOT    P00143	// R_1st DIE FPCB ALIGN FWD/BWD
AND LOAD
LOAD NOT  P00063	// R_1st DIE FPCB ALIGN FORWARD
AND NOT   T1068	// R_1st DIE FPCB ALIGN BACKWARD
OR LOAD
TON       T0571 400	// R_1st DIE FPCB FWD/BWD SN ALARM
; L322
LOAD      M00718	// R_1st DIE FPCB FWD/BWD SN ALARM
AND NOT   M00008	// LEFT RESET SW PLS
OR        T0571	// R_1st DIE FPCB FWD/BWD SN ALARM
OUT       M00718	// R_1st DIE FPCB FWD/BWD SN ALARM
; L324
LOAD      P00064	// R_1-1 ROTATE MANDREL FORWARD
OR        P00144	// R_1-1 ROTATE FWD/BWD
LOAD      P00065	// R_1-1 ROTATE MANDREL BACKWARD
OR NOT    P00144	// R_1-1 ROTATE FWD/BWD
AND LOAD
LOAD NOT  P00064	// R_1-1 ROTATE MANDREL FORWARD
AND NOT   P00065	// R_1-1 ROTATE MANDREL BACKWARD
OR LOAD
TON       T0572 400	// R_1st MAND FWD/BWD SN ALARM

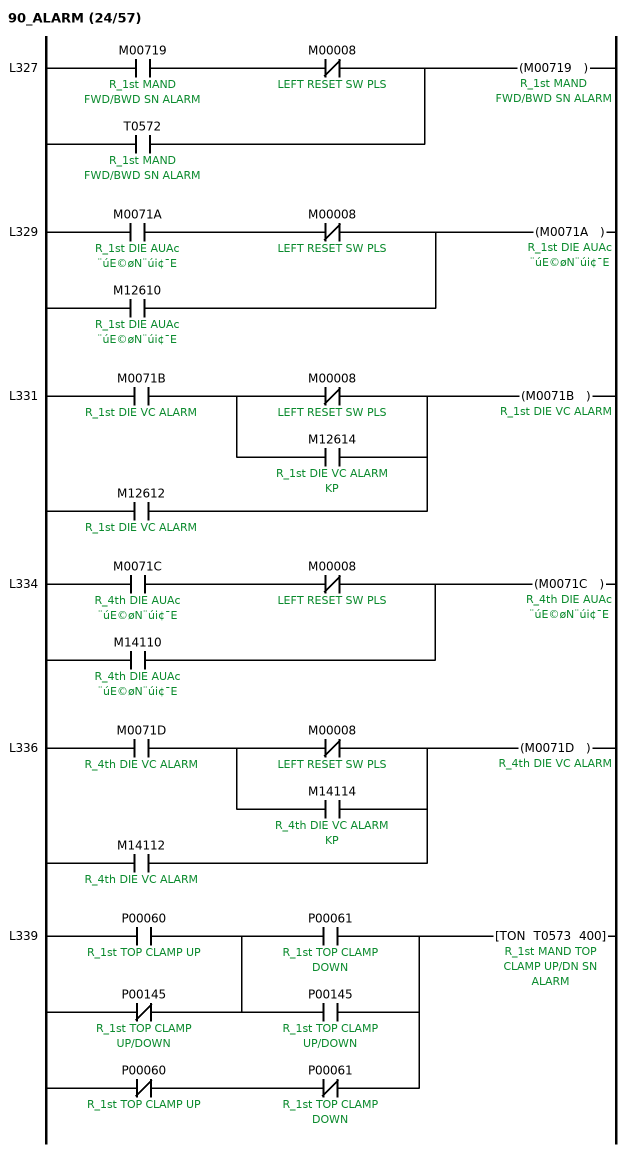
; L327
LOAD      M00719	// R_1st MAND FWD/BWD SN ALARM
AND NOT   M00008	// LEFT RESET SW PLS
OR        T0572	// R_1st MAND FWD/BWD SN ALARM
OUT       M00719	// R_1st MAND FWD/BWD SN ALARM
; L329
LOAD      M0071A	// R_1st DIE AUAc ¨úE©øN¨úi¢¯E
AND NOT   M00008	// LEFT RESET SW PLS
OR        M12610	// R_1st DIE AUAc ¨úE©øN¨úi¢¯E
OUT       M0071A	// R_1st DIE AUAc ¨úE©øN¨úi¢¯E
; L331
LOAD      M0071B	// R_1st DIE VC ALARM
LOAD NOT  M00008	// LEFT RESET SW PLS
OR        M12614	// R_1st DIE VC ALARM KP
AND LOAD
OR        M12612	// R_1st DIE VC ALARM
OUT       M0071B	// R_1st DIE VC ALARM
; L334
LOAD      M0071C	// R_4th DIE AUAc ¨úE©øN¨úi¢¯E
AND NOT   M00008	// LEFT RESET SW PLS
OR        M14110	// R_4th DIE AUAc ¨úE©øN¨úi¢¯E
OUT       M0071C	// R_4th DIE AUAc ¨úE©øN¨úi¢¯E
; L336
LOAD      M0071D	// R_4th DIE VC ALARM
LOAD NOT  M00008	// LEFT RESET SW PLS
OR        M14114	// R_4th DIE VC ALARM KP
AND LOAD
OR        M14112	// R_4th DIE VC ALARM
OUT       M0071D	// R_4th DIE VC ALARM
; L339
LOAD      P00060	// R_1st TOP CLAMP UP
OR NOT    P00145	// R_1st TOP CLAMP UP/DOWN
LOAD      P00061	// R_1st TOP CLAMP DOWN
OR        P00145	// R_1st TOP CLAMP UP/DOWN
AND LOAD
LOAD NOT  P00060	// R_1st TOP CLAMP UP
AND NOT   P00061	// R_1st TOP CLAMP DOWN
OR LOAD
TON       T0573 400	// R_1st MAND TOP CLAMP UP/DN SN ALARM

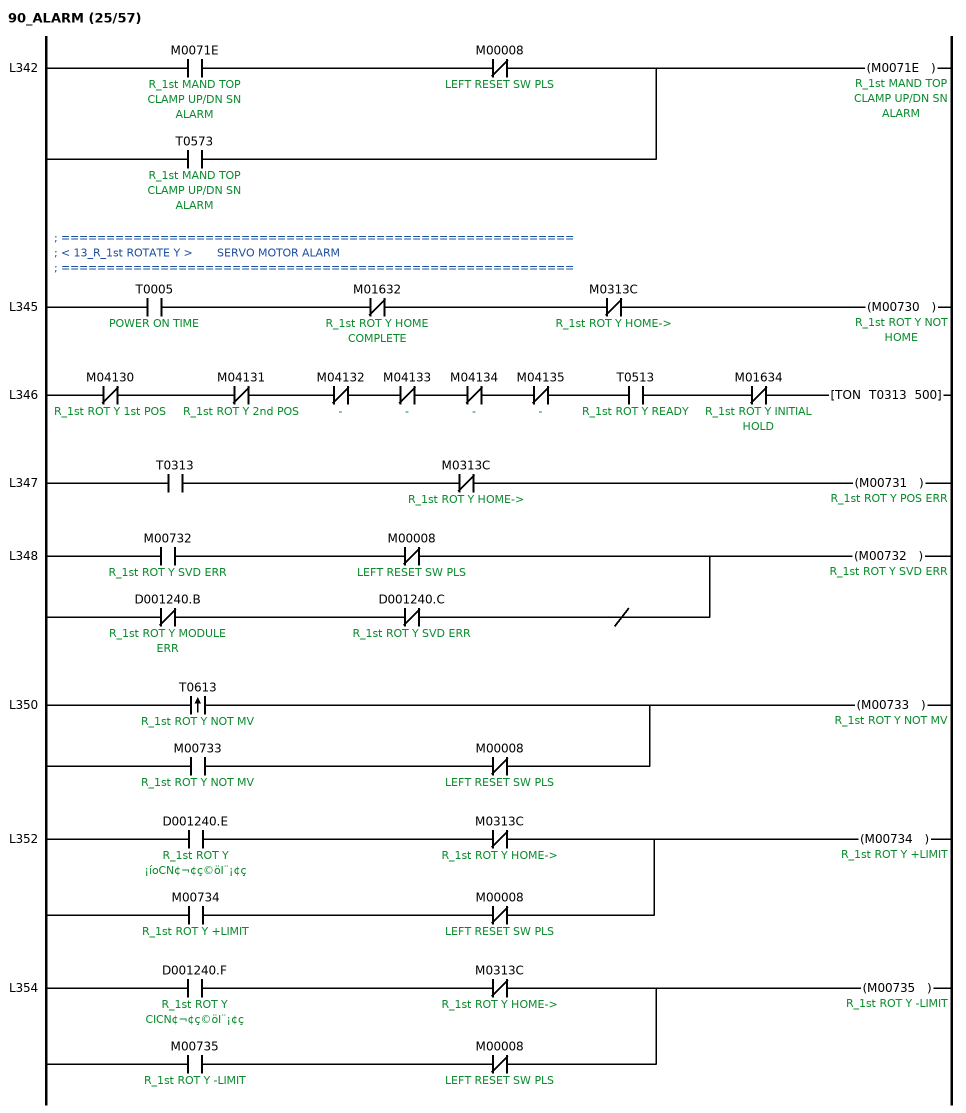
; L342
LOAD      M0071E	// R_1st MAND TOP CLAMP UP/DN SN ALARM
AND NOT   M00008	// LEFT RESET SW PLS
OR        T0573	// R_1st MAND TOP CLAMP UP/DN SN ALARM
OUT       M0071E	// R_1st MAND TOP CLAMP UP/DN SN ALARM
// =========================================================
// 
//        < 13_R_1st ROTATE Y >       SERVO MOTOR ALARM
// 
// =========================================================
; L345
LOAD      T0005	// POWER ON TIME
AND NOT   M01632	// R_1st ROT Y HOME COMPLETE
AND NOT   M0313C	// R_1st ROT Y HOME->
OUT       M00730	// R_1st ROT Y NOT HOME
; L346
LOAD NOT  M04130	// R_1st ROT Y 1st POS
AND NOT   M04131	// R_1st ROT Y 2nd POS
AND NOT   M04132	// -
AND NOT   M04133	// -
AND NOT   M04134	// -
AND NOT   M04135	// -
AND       T0513	// R_1st ROT Y READY
AND NOT   M01634	// R_1st ROT Y INITIAL HOLD
TON       T0313 500
; L347
LOAD      T0313
AND NOT   M0313C	// R_1st ROT Y HOME->
OUT       M00731	// R_1st ROT Y POS ERR
; L348
LOAD      M00732	// R_1st ROT Y SVD ERR
AND NOT   M00008	// LEFT RESET SW PLS
LOAD NOT  D001240.B	// R_1st ROT Y MODULE ERR
AND NOT   D001240.C	// R_1st ROT Y SVD ERR
NOT
OR LOAD
OUT       M00732	// R_1st ROT Y SVD ERR
; L350
LOADP     T0613	// R_1st ROT Y NOT MV
LOAD      M00733	// R_1st ROT Y NOT MV
AND NOT   M00008	// LEFT RESET SW PLS
OR LOAD
OUT       M00733	// R_1st ROT Y NOT MV
; L352
LOAD      D001240.E	// R_1st ROT Y ¡íoCN¢¬¢ç©öI¨¡¢ç
AND NOT   M0313C	// R_1st ROT Y HOME->
LOAD      M00734	// R_1st ROT Y +LIMIT
AND NOT   M00008	// LEFT RESET SW PLS
OR LOAD
OUT       M00734	// R_1st ROT Y +LIMIT
; L354
LOAD      D001240.F	// R_1st ROT Y CICN¢¬¢ç©öI¨¡¢ç
AND NOT   M0313C	// R_1st ROT Y HOME->
LOAD      M00735	// R_1st ROT Y -LIMIT
AND NOT   M00008	// LEFT RESET SW PLS
OR LOAD
OUT       M00735	// R_1st ROT Y -LIMIT

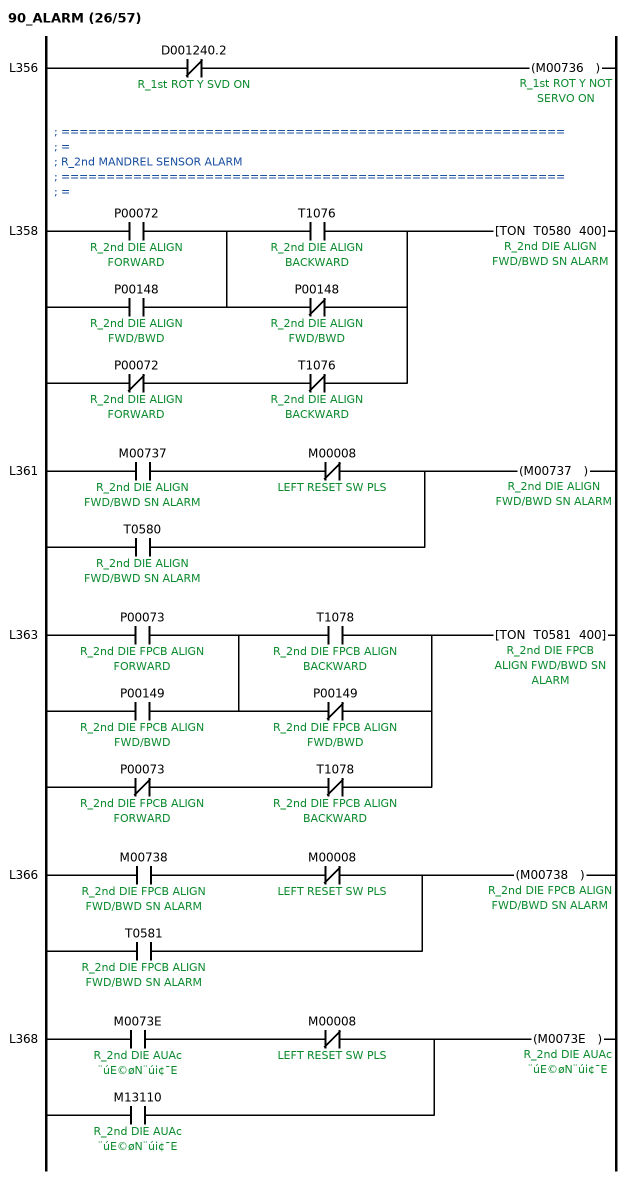
; L356
LOAD NOT  D001240.2	// R_1st ROT Y SVD ON
OUT       M00736	// R_1st ROT Y NOT SERVO ON
// =========================================================
// 
//        R_2nd MANDREL SENSOR ALARM
// 
// =========================================================
; L358
LOAD      P00072	// R_2nd DIE ALIGN FORWARD
OR        P00148	// R_2nd DIE ALIGN FWD/BWD
LOAD      T1076	// R_2nd DIE ALIGN BACKWARD
OR NOT    P00148	// R_2nd DIE ALIGN FWD/BWD
AND LOAD
LOAD NOT  P00072	// R_2nd DIE ALIGN FORWARD
AND NOT   T1076	// R_2nd DIE ALIGN BACKWARD
OR LOAD
TON       T0580 400	// R_2nd DIE ALIGN FWD/BWD SN ALARM
; L361
LOAD      M00737	// R_2nd DIE ALIGN FWD/BWD SN ALARM
AND NOT   M00008	// LEFT RESET SW PLS
OR        T0580	// R_2nd DIE ALIGN FWD/BWD SN ALARM
OUT       M00737	// R_2nd DIE ALIGN FWD/BWD SN ALARM
; L363
LOAD      P00073	// R_2nd DIE FPCB ALIGN FORWARD
OR        P00149	// R_2nd DIE FPCB ALIGN FWD/BWD
LOAD      T1078	// R_2nd DIE FPCB ALIGN BACKWARD
OR NOT    P00149	// R_2nd DIE FPCB ALIGN FWD/BWD
AND LOAD
LOAD NOT  P00073	// R_2nd DIE FPCB ALIGN FORWARD
AND NOT   T1078	// R_2nd DIE FPCB ALIGN BACKWARD
OR LOAD
TON       T0581 400	// R_2nd DIE FPCB ALIGN FWD/BWD SN ALARM
; L366
LOAD      M00738	// R_2nd DIE FPCB ALIGN FWD/BWD SN ALARM
AND NOT   M00008	// LEFT RESET SW PLS
OR        T0581	// R_2nd DIE FPCB ALIGN FWD/BWD SN ALARM
OUT       M00738	// R_2nd DIE FPCB ALIGN FWD/BWD SN ALARM
; L368
LOAD      M0073E	// R_2nd DIE AUAc ¨úE©øN¨úi¢¯E
AND NOT   M00008	// LEFT RESET SW PLS
OR        M13110	// R_2nd DIE AUAc ¨úE©øN¨úi¢¯E
OUT       M0073E	// R_2nd DIE AUAc ¨úE©øN¨úi¢¯E

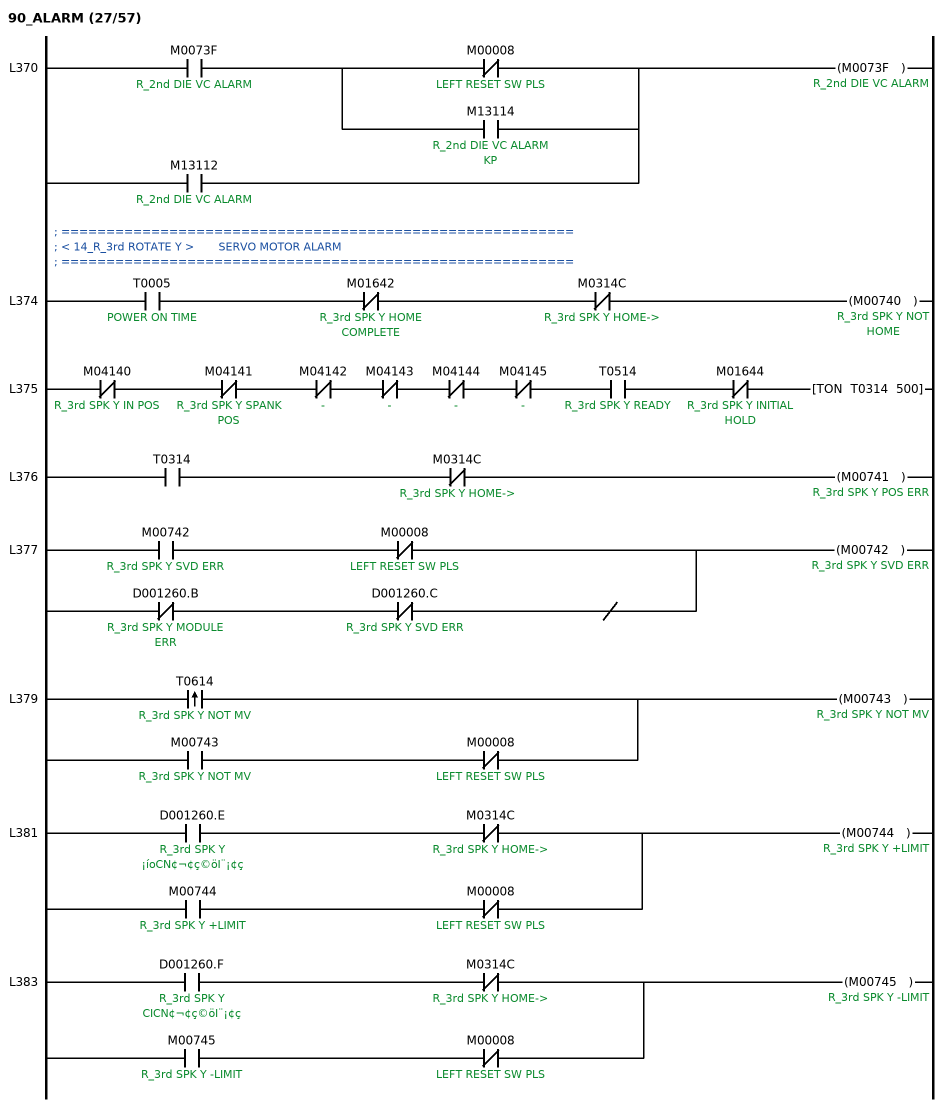
; L370
LOAD      M0073F	// R_2nd DIE VC ALARM
LOAD NOT  M00008	// LEFT RESET SW PLS
OR        M13114	// R_2nd DIE VC ALARM KP
AND LOAD
OR        M13112	// R_2nd DIE VC ALARM
OUT       M0073F	// R_2nd DIE VC ALARM
// =========================================================
// 
//        < 14_R_3rd ROTATE Y >       SERVO MOTOR ALARM
// 
// =========================================================
; L374
LOAD      T0005	// POWER ON TIME
AND NOT   M01642	// R_3rd SPK Y HOME COMPLETE
AND NOT   M0314C	// R_3rd SPK Y HOME->
OUT       M00740	// R_3rd SPK Y NOT HOME
; L375
LOAD NOT  M04140	// R_3rd SPK Y IN POS
AND NOT   M04141	// R_3rd SPK Y SPANK POS
AND NOT   M04142	// -
AND NOT   M04143	// -
AND NOT   M04144	// -
AND NOT   M04145	// -
AND       T0514	// R_3rd SPK Y READY
AND NOT   M01644	// R_3rd SPK Y INITIAL HOLD
TON       T0314 500
; L376
LOAD      T0314
AND NOT   M0314C	// R_3rd SPK Y HOME->
OUT       M00741	// R_3rd SPK Y POS ERR
; L377
LOAD      M00742	// R_3rd SPK Y SVD ERR
AND NOT   M00008	// LEFT RESET SW PLS
LOAD NOT  D001260.B	// R_3rd SPK Y MODULE ERR
AND NOT   D001260.C	// R_3rd SPK Y SVD ERR
NOT
OR LOAD
OUT       M00742	// R_3rd SPK Y SVD ERR
; L379
LOADP     T0614	// R_3rd SPK Y NOT MV
LOAD      M00743	// R_3rd SPK Y NOT MV
AND NOT   M00008	// LEFT RESET SW PLS
OR LOAD
OUT       M00743	// R_3rd SPK Y NOT MV
; L381
LOAD      D001260.E	// R_3rd SPK Y ¡íoCN¢¬¢ç©öI¨¡¢ç
AND NOT   M0314C	// R_3rd SPK Y HOME->
LOAD      M00744	// R_3rd SPK Y +LIMIT
AND NOT   M00008	// LEFT RESET SW PLS
OR LOAD
OUT       M00744	// R_3rd SPK Y +LIMIT
; L383
LOAD      D001260.F	// R_3rd SPK Y CICN¢¬¢ç©öI¨¡¢ç
AND NOT   M0314C	// R_3rd SPK Y HOME->
LOAD      M00745	// R_3rd SPK Y -LIMIT
AND NOT   M00008	// LEFT RESET SW PLS
OR LOAD
OUT       M00745	// R_3rd SPK Y -LIMIT

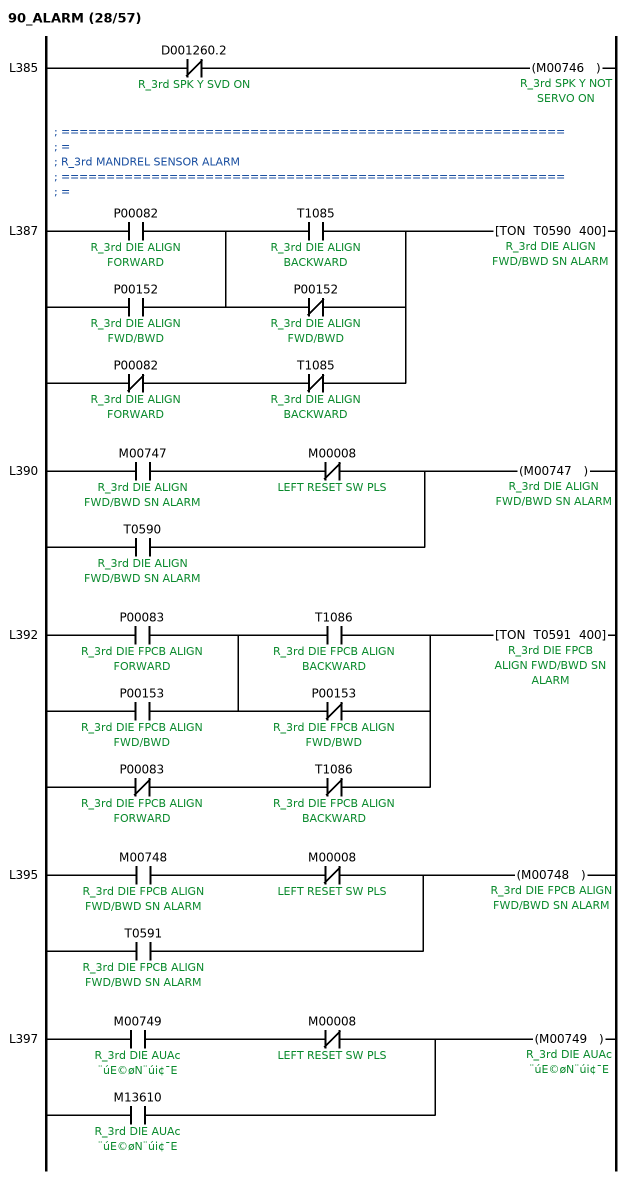
; L385
LOAD NOT  D001260.2	// R_3rd SPK Y SVD ON
OUT       M00746	// R_3rd SPK Y NOT SERVO ON
// =========================================================
// 
//        R_3rd MANDREL SENSOR ALARM
// 
// =========================================================
; L387
LOAD      P00082	// R_3rd DIE ALIGN FORWARD
OR        P00152	// R_3rd DIE ALIGN FWD/BWD
LOAD      T1085	// R_3rd DIE ALIGN BACKWARD
OR NOT    P00152	// R_3rd DIE ALIGN FWD/BWD
AND LOAD
LOAD NOT  P00082	// R_3rd DIE ALIGN FORWARD
AND NOT   T1085	// R_3rd DIE ALIGN BACKWARD
OR LOAD
TON       T0590 400	// R_3rd DIE ALIGN FWD/BWD SN ALARM
; L390
LOAD      M00747	// R_3rd DIE ALIGN FWD/BWD SN ALARM
AND NOT   M00008	// LEFT RESET SW PLS
OR        T0590	// R_3rd DIE ALIGN FWD/BWD SN ALARM
OUT       M00747	// R_3rd DIE ALIGN FWD/BWD SN ALARM
; L392
LOAD      P00083	// R_3rd DIE FPCB ALIGN FORWARD
OR        P00153	// R_3rd DIE FPCB ALIGN FWD/BWD
LOAD      T1086	// R_3rd DIE FPCB ALIGN BACKWARD
OR NOT    P00153	// R_3rd DIE FPCB ALIGN FWD/BWD
AND LOAD
LOAD NOT  P00083	// R_3rd DIE FPCB ALIGN FORWARD
AND NOT   T1086	// R_3rd DIE FPCB ALIGN BACKWARD
OR LOAD
TON       T0591 400	// R_3rd DIE FPCB ALIGN FWD/BWD SN ALARM
; L395
LOAD      M00748	// R_3rd DIE FPCB ALIGN FWD/BWD SN ALARM
AND NOT   M00008	// LEFT RESET SW PLS
OR        T0591	// R_3rd DIE FPCB ALIGN FWD/BWD SN ALARM
OUT       M00748	// R_3rd DIE FPCB ALIGN FWD/BWD SN ALARM
; L397
LOAD      M00749	// R_3rd DIE AUAc ¨úE©øN¨úi¢¯E
AND NOT   M00008	// LEFT RESET SW PLS
OR        M13610	// R_3rd DIE AUAc ¨úE©øN¨úi¢¯E
OUT       M00749	// R_3rd DIE AUAc ¨úE©øN¨úi¢¯E

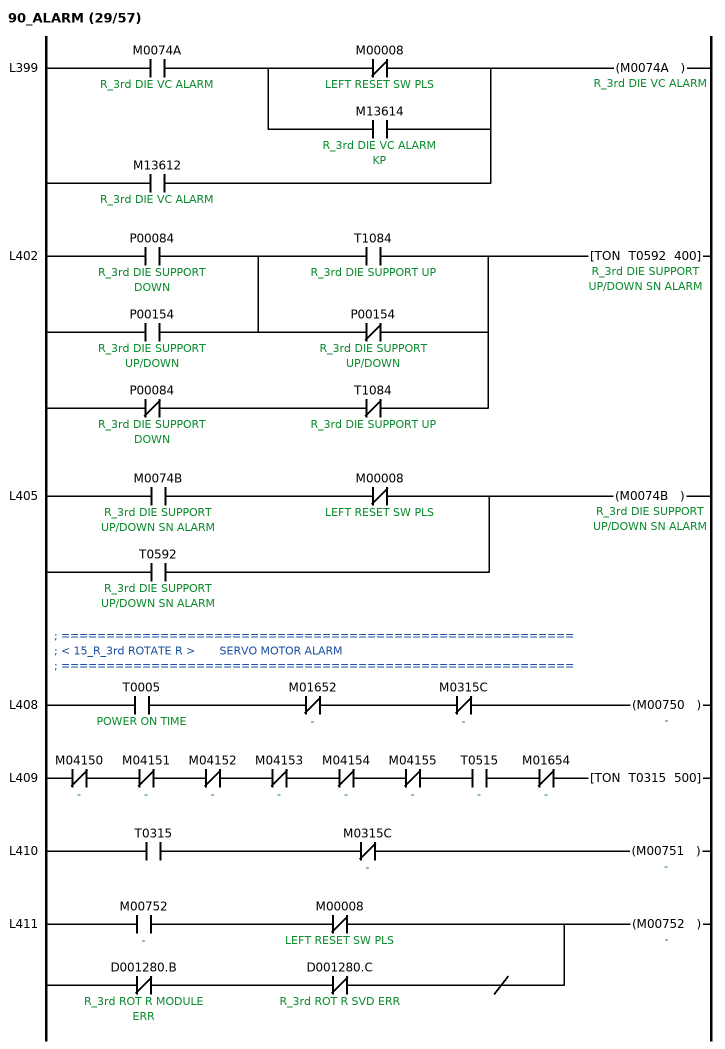
; L399
LOAD      M0074A	// R_3rd DIE VC ALARM
LOAD NOT  M00008	// LEFT RESET SW PLS
OR        M13614	// R_3rd DIE VC ALARM KP
AND LOAD
OR        M13612	// R_3rd DIE VC ALARM
OUT       M0074A	// R_3rd DIE VC ALARM
; L402
LOAD      P00084	// R_3rd DIE SUPPORT DOWN
OR        P00154	// R_3rd DIE SUPPORT UP/DOWN
LOAD      T1084	// R_3rd DIE SUPPORT UP
OR NOT    P00154	// R_3rd DIE SUPPORT UP/DOWN
AND LOAD
LOAD NOT  P00084	// R_3rd DIE SUPPORT DOWN
AND NOT   T1084	// R_3rd DIE SUPPORT UP
OR LOAD
TON       T0592 400	// R_3rd DIE SUPPORT UP/DOWN SN ALARM
; L405
LOAD      M0074B	// R_3rd DIE SUPPORT UP/DOWN SN ALARM
AND NOT   M00008	// LEFT RESET SW PLS
OR        T0592	// R_3rd DIE SUPPORT UP/DOWN SN ALARM
OUT       M0074B	// R_3rd DIE SUPPORT UP/DOWN SN ALARM
// =========================================================
// 
//        < 15_R_3rd ROTATE R >       SERVO MOTOR ALARM
// 
// =========================================================
; L408
LOAD      T0005	// POWER ON TIME
AND NOT   M01652	// -
AND NOT   M0315C	// -
OUT       M00750	// -
; L409
LOAD NOT  M04150	// -
AND NOT   M04151	// -
AND NOT   M04152	// -
AND NOT   M04153	// -
AND NOT   M04154	// -
AND NOT   M04155	// -
AND       T0515	// -
AND NOT   M01654	// -
TON       T0315 500
; L410
LOAD      T0315
AND NOT   M0315C	// -
OUT       M00751	// -
; L411
LOAD      M00752	// -
AND NOT   M00008	// LEFT RESET SW PLS
LOAD NOT  D001280.B	// R_3rd ROT R MODULE ERR
AND NOT   D001280.C	// R_3rd ROT R SVD ERR
NOT
OR LOAD
OUT       M00752	// -

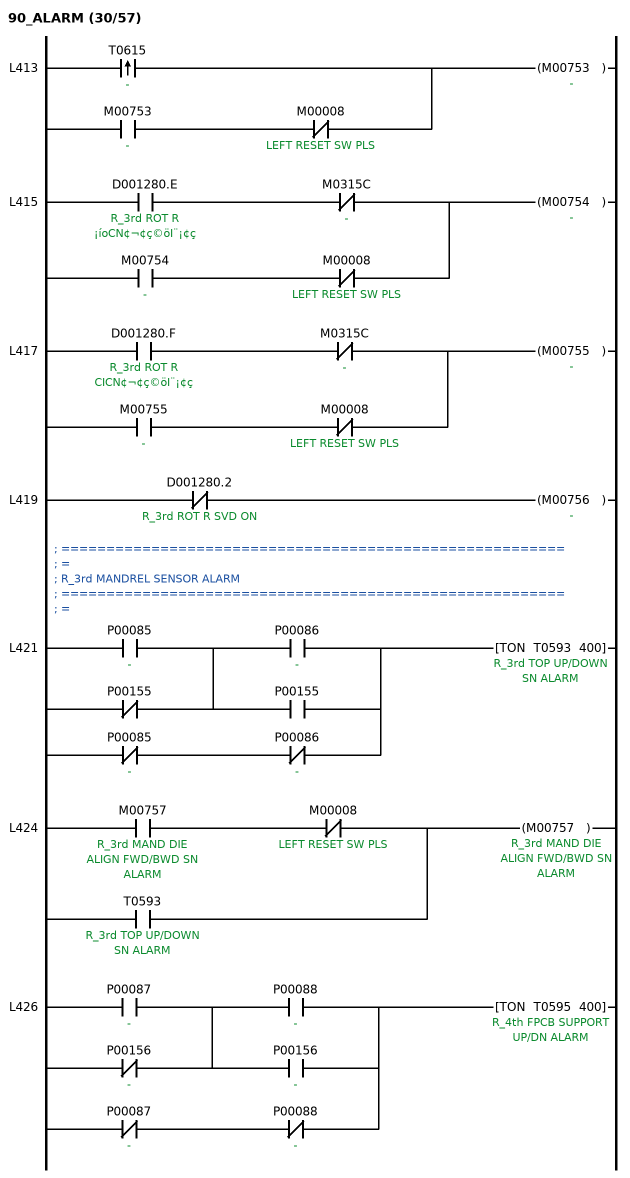
; L413
LOADP     T0615	// -
LOAD      M00753	// -
AND NOT   M00008	// LEFT RESET SW PLS
OR LOAD
OUT       M00753	// -
; L415
LOAD      D001280.E	// R_3rd ROT R ¡íoCN¢¬¢ç©öI¨¡¢ç
AND NOT   M0315C	// -
LOAD      M00754	// -
AND NOT   M00008	// LEFT RESET SW PLS
OR LOAD
OUT       M00754	// -
; L417
LOAD      D001280.F	// R_3rd ROT R CICN¢¬¢ç©öI¨¡¢ç
AND NOT   M0315C	// -
LOAD      M00755	// -
AND NOT   M00008	// LEFT RESET SW PLS
OR LOAD
OUT       M00755	// -
; L419
LOAD NOT  D001280.2	// R_3rd ROT R SVD ON
OUT       M00756	// -
// =========================================================
// 
//        R_3rd MANDREL SENSOR ALARM
// 
// =========================================================
; L421
LOAD      P00085	// -
OR NOT    P00155
LOAD      P00086	// -
OR        P00155
AND LOAD
LOAD NOT  P00085	// -
AND NOT   P00086	// -
OR LOAD
TON       T0593 400	// R_3rd TOP UP/DOWN SN ALARM
; L424
LOAD      M00757	// R_3rd MAND DIE ALIGN FWD/BWD SN ALARM
AND NOT   M00008	// LEFT RESET SW PLS
OR        T0593	// R_3rd TOP UP/DOWN SN ALARM
OUT       M00757	// R_3rd MAND DIE ALIGN FWD/BWD SN ALARM
; L426
LOAD      P00087	// -
OR NOT    P00156	// -
LOAD      P00088	// -
OR        P00156	// -
AND LOAD
LOAD NOT  P00087	// -
AND NOT   P00088	// -
OR LOAD
TON       T0595 400	// R_4th FPCB SUPPORT UP/DN ALARM

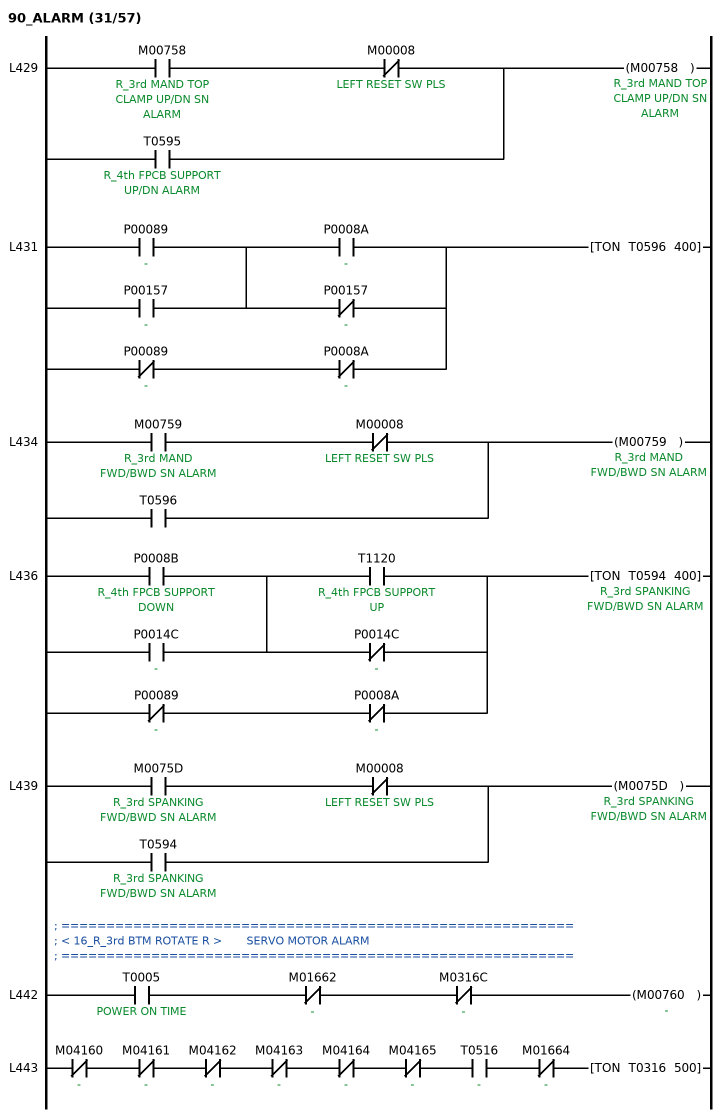
; L429
LOAD      M00758	// R_3rd MAND TOP CLAMP UP/DN SN ALARM
AND NOT   M00008	// LEFT RESET SW PLS
OR        T0595	// R_4th FPCB SUPPORT UP/DN ALARM
OUT       M00758	// R_3rd MAND TOP CLAMP UP/DN SN ALARM
; L431
LOAD      P00089	// -
OR        P00157	// -
LOAD      P0008A	// -
OR NOT    P00157	// -
AND LOAD
LOAD NOT  P00089	// -
AND NOT   P0008A	// -
OR LOAD
TON       T0596 400
; L434
LOAD      M00759	// R_3rd MAND FWD/BWD SN ALARM
AND NOT   M00008	// LEFT RESET SW PLS
OR        T0596
OUT       M00759	// R_3rd MAND FWD/BWD SN ALARM
; L436
LOAD      P0008B	// R_4th FPCB SUPPORT DOWN
OR        P0014C	// -
LOAD      T1120	// R_4th FPCB SUPPORT UP
OR NOT    P0014C	// -
AND LOAD
LOAD NOT  P00089	// -
AND NOT   P0008A	// -
OR LOAD
TON       T0594 400	// R_3rd SPANKING FWD/BWD SN ALARM
; L439
LOAD      M0075D	// R_3rd SPANKING FWD/BWD SN ALARM
AND NOT   M00008	// LEFT RESET SW PLS
OR        T0594	// R_3rd SPANKING FWD/BWD SN ALARM
OUT       M0075D	// R_3rd SPANKING FWD/BWD SN ALARM
// =========================================================
// 
//        < 16_R_3rd BTM ROTATE R >       SERVO MOTOR ALARM
// 
// =========================================================
; L442
LOAD      T0005	// POWER ON TIME
AND NOT   M01662	// -
AND NOT   M0316C	// -
OUT       M00760	// -
; L443
LOAD NOT  M04160	// -
AND NOT   M04161	// -
AND NOT   M04162	// -
AND NOT   M04163	// -
AND NOT   M04164	// -
AND NOT   M04165	// -
AND       T0516	// -
AND NOT   M01664	// -
TON       T0316 500

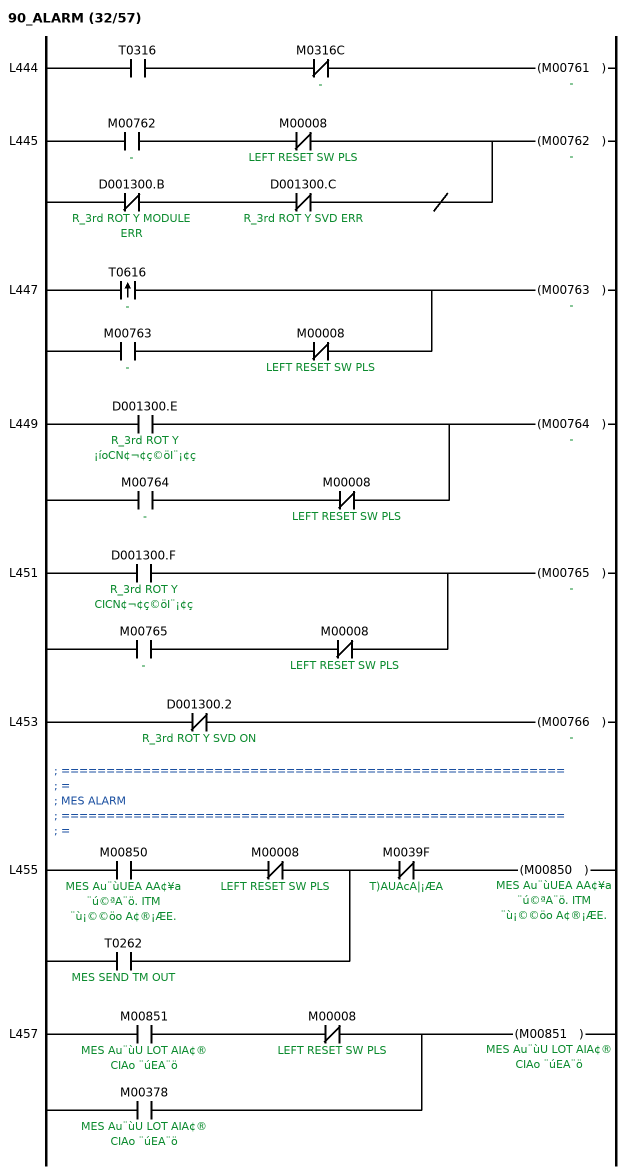
; L444
LOAD      T0316
AND NOT   M0316C	// -
OUT       M00761	// -
; L445
LOAD      M00762	// -
AND NOT   M00008	// LEFT RESET SW PLS
LOAD NOT  D001300.B	// R_3rd ROT Y MODULE ERR
AND NOT   D001300.C	// R_3rd ROT Y SVD ERR
NOT
OR LOAD
OUT       M00762	// -
; L447
LOADP     T0616	// -
LOAD      M00763	// -
AND NOT   M00008	// LEFT RESET SW PLS
OR LOAD
OUT       M00763	// -
; L449
LOAD      D001300.E	// R_3rd ROT Y ¡íoCN¢¬¢ç©öI¨¡¢ç
LOAD      M00764	// -
AND NOT   M00008	// LEFT RESET SW PLS
OR LOAD
OUT       M00764	// -
; L451
LOAD      D001300.F	// R_3rd ROT Y CICN¢¬¢ç©öI¨¡¢ç
LOAD      M00765	// -
AND NOT   M00008	// LEFT RESET SW PLS
OR LOAD
OUT       M00765	// -
; L453
LOAD NOT  D001300.2	// R_3rd ROT Y SVD ON
OUT       M00766	// -
// =========================================================
// 
//        MES ALARM
// 
// =========================================================
; L455
LOAD      M00850	// MES Au¨ùUEA AA¢¥a ¨ú©ªA¨ö. ITM ¨ù¡©©öo A¢®¡ÆE.
AND NOT   M00008	// LEFT RESET SW PLS
OR        T0262	// MES SEND TM OUT
AND NOT   M0039F	// T)AUAcA|¡ÆA
OUT       M00850	// MES Au¨ùUEA AA¢¥a ¨ú©ªA¨ö. ITM ¨ù¡©©öo A¢®¡ÆE.
; L457
LOAD      M00851	// MES Au¨ùU LOT AIA¢® CIAo ¨úEA¨ö
AND NOT   M00008	// LEFT RESET SW PLS
OR        M00378	// MES Au¨ùU LOT AIA¢® CIAo ¨úEA¨ö
OUT       M00851	// MES Au¨ùU LOT AIA¢® CIAo ¨úEA¨ö

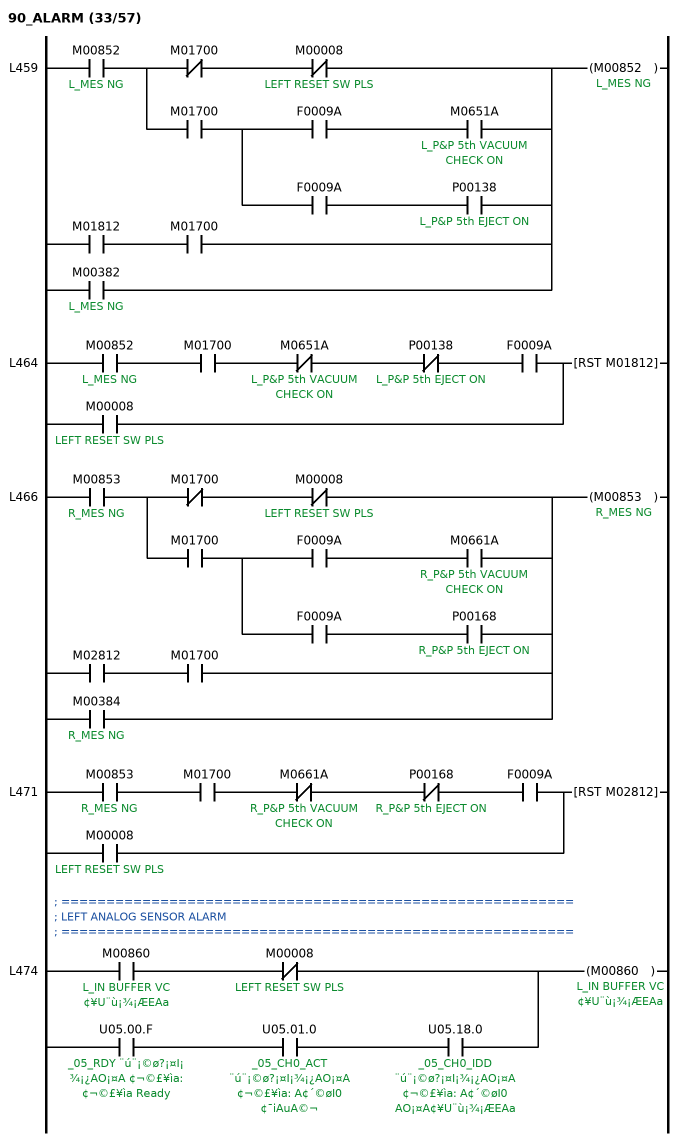
; L459
LOAD      M00852	// L_MES NG
LOAD NOT  M01700
AND NOT   M00008	// LEFT RESET SW PLS
LOAD      M01700
LOAD      F0009A
AND       M0651A	// L_P&P 5th VACUUM CHECK ON
LOAD      F0009A
AND       P00138	// L_P&P 5th EJECT ON
OR LOAD
AND LOAD
OR LOAD
AND LOAD
LOAD      M01812
AND       M01700
OR LOAD
OR        M00382	// L_MES NG
OUT       M00852	// L_MES NG
; L464
LOAD      M00852	// L_MES NG
AND       M01700
AND NOT   M0651A	// L_P&P 5th VACUUM CHECK ON
AND NOT   P00138	// L_P&P 5th EJECT ON
AND       F0009A
OR        M00008	// LEFT RESET SW PLS
RST       M01812
; L466
LOAD      M00853	// R_MES NG
LOAD NOT  M01700
AND NOT   M00008	// LEFT RESET SW PLS
LOAD      M01700
LOAD      F0009A
AND       M0661A	// R_P&P 5th VACUUM CHECK ON
LOAD      F0009A
AND       P00168	// R_P&P 5th EJECT ON
OR LOAD
AND LOAD
OR LOAD
AND LOAD
LOAD      M02812
AND       M01700
OR LOAD
OR        M00384	// R_MES NG
OUT       M00853	// R_MES NG
; L471
LOAD      M00853	// R_MES NG
AND       M01700
AND NOT   M0661A	// R_P&P 5th VACUUM CHECK ON
AND NOT   P00168	// R_P&P 5th EJECT ON
AND       F0009A
OR        M00008	// LEFT RESET SW PLS
RST       M02812
// =========================================================
// 
//        LEFT ANALOG SENSOR ALARM
// 
// =========================================================
; L474
LOAD      M00860	// L_IN BUFFER VC ¢¥U¨ù¡¾¡ÆEAa
AND NOT   M00008	// LEFT RESET SW PLS
LOAD      U05.00.F	// _05_RDY ¨ú¨¡©ø?¡¤I¡¾¡¿AO¡¤A ¢¬©£¥ìa: ¢¬©£¥ìa Ready
AND       U05.01.0	// _05_CH0_ACT ¨ú¨¡©ø?¡¤I¡¾¡¿AO¡¤A ¢¬©£¥ìa: A¢´©øI0 ¢¯iAuA©¬
AND       U05.18.0	// _05_CH0_IDD ¨ú¨¡©ø?¡¤I¡¾¡¿AO¡¤A ¢¬©£¥ìa: A¢´©øI0 AO¡¤A¢¥U¨ù¡¾¡ÆEAa
OR LOAD
OUT       M00860	// L_IN BUFFER VC ¢¥U¨ù¡¾¡ÆEAa

